LIN {X 0,Y 352.522,Z 1249.974,A -85,B 0,C 180,E1 16301.444,E2 16301.444} C_VEL
LIN {X 0,Y 352.114,Z 1252.721,A -85,B 0,C 180,E1 16297.99,E2 16297.99} C_VEL
LIN {X 0,Y 351.998,Z 1254.362,A -85,B 0,C 180,E1 16294.881,E2 16294.881} C_VEL
LIN {X 0,Y 351.964,Z 1255.218,A -85,B 0,C 180,E1 16291.783,E2 16291.783} C_VEL
LIN {X 0,Y 351.944,Z 1255.295,A -85,B 0,C 180,E1 16288.69,E2 16288.69} C_VEL
LIN {X 0,Y 351.993,Z 1254.526,A -85,B 0,C 180,E1 16285.431,E2 16285.431} C_VEL
LIN {X 0,Y 352.107,Z 1252.886,A -85,B 0,C 180,E1 16282.159,E2 16282.159} C_VEL
LIN {X 0,Y 352.483,Z 1250.205,A -85,B 0,C 180,E1 16278.706,E2 16278.706} C_VEL
LIN {X 0,Y 353.184,Z 1246.726,A -85,B 0,C 180,E1 16275.399,E2 16275.399} C_VEL
LIN {X 0,Y 354.443,Z 1242.064,A -85,B 0,C 180,E1 16271.915,E2 16271.915} C_VEL
LIN {X 0,Y 356.359,Z 1236.339,A -85,B 0,C 180,E1 16268.428,E2 16268.428} C_VEL
LIN {X 0,Y 359.376,Z 1228.818,A -85,B 0,C 180,E1 16264.623,E2 16264.623} C_VEL
LIN {X 0,Y 362.896,Z 1220.993,A -85,B 0,C 180,E1 16261.294,E2 16261.294} C_VEL
LIN {X 0,Y 363.326,Z 1218.334,A -85,B 0,C 180,E1 16260.145,E2 16260.145} C_VEL
LIN {X 0,Y 361.437,Z 1211.116,A -85,B 0,C 180,E1 16256.998,E2 16256.998} C_VEL
LIN {X 0,Y 362.2,Z 1208.382,A -85,B 0,C 180,E1 16256.041,E2 16256.041} C_VEL
LIN {X 0,Y 367.884,Z 1197.913,A -85,B 0,C 180,E1 16252.881,E2 16252.881} C_VEL
LIN {X 0,Y 374.556,Z 1185.938,A -85,B 0,C 180,E1 16249.751,E2 16249.751} C_VEL
LIN {X 0,Y 384.203,Z 1168.784,A -85,B 0,C 180,E1 16245.977,E2 16245.977} C_VEL
LIN {X 0,Y 392.178,Z 1154.367,A -85,B 0,C 180,E1 16243.302,E2 16243.302} C_VEL
LIN {X 0,Y 399.981,Z 1139.957,A -85,B 0,C 180,E1 16240.973,E2 16240.973} C_VEL
LIN {X 0,Y 408.048,Z 1124.586,A -85,B 0,C 180,E1 16238.804,E2 16238.804} C_VEL
LIN {X 0,Y 418.139,Z 1104.607,A -85,B 0,C 180,E1 16236.373,E2 16236.373} C_VEL
LIN {X 0,Y 427.575,Z 1084.304,A -85,B 0,C 180,E1 16234.304,E2 16234.304} C_VEL
LIN {X 0,Y 435.512,Z 1066.092,A -85,B 0,C 180,E1 16232.701,E2 16232.701} C_VEL
LIN {X 0,Y 442.95,Z 1047.765,A -85,B 0,C 180,E1 16231.3,E2 16231.3} C_VEL
LIN {X 0,Y 449.994,Z 1028.988,A -85,B 0,C 180,E1 16230.058,E2 16230.058} C_VEL
LIN {X 0,Y 457.896,Z 1005.714,A -85,B 0,C 180,E1 16228.73,E2 16228.73} C_VEL
LIN {X 0,Y 465.26,Z 980.582,A -85,B 0,C 180,E1 16227.557,E2 16227.557} C_VEL
LIN {X 0,Y 470.568,Z 959.738,A -85,B 0,C 180,E1 16226.745,E2 16226.745} C_VEL
LIN {X 0,Y 475.18,Z 938.773,A -85,B 0,C 180,E1 16226.067,E2 16226.067} C_VEL
LIN {X 0,Y 479.078,Z 917.527,A -85,B 0,C 180,E1 16225.5,E2 16225.5} C_VEL
LIN {X 0,Y 482.827,Z 891.865,A -85,B 0,C 180,E1 16224.963,E2 16224.963} C_VEL
LIN {X 0,Y 486.213,Z 853.496,A -85,B 0,C 180,E1 16224.337,E2 16224.337} C_VEL
LIN {X 0,Y 503.252,Z 634.163,A -85,B 0,C 180,E1 16220.941,E2 16220.941} C_VEL
LIN {X 0,Y 505.06,Z 611.125,A -85,B 0,C 180,E1 16220.573,E2 16220.573} C_VEL
LIN {X 0,Y 498.511,Z 600.707,A -85,B 0,C 180,E1 16217.962,E2 16217.962} C_VEL
LIN {X 0,Y 493.261,Z 592.705,A -85,B 0,C 180,E1 16215.52,E2 16215.52} C_VEL
LIN {X 0,Y 490.584,Z 588.712,A -85,B 0,C 180,E1 16214.097,E2 16214.097} C_VEL
LIN {X 0,Y 487.897,Z 584.679,A -85,B 0,C 180,E1 16212.487,E2 16212.487} C_VEL
LIN {X 0,Y 484.928,Z 580.257,A -85,B 0,C 180,E1 16210.398,E2 16210.398} C_VEL
LIN {X 0,Y 482.057,Z 575.835,A -85,B 0,C 180,E1 16207.808,E2 16207.808} C_VEL
LIN {X 0,Y 478.927,Z 571.053,A -85,B 0,C 180,E1 16202.872,E2 16202.872} C_VEL
LIN {X 0,Y 478.709,Z 569.893,A -85,B 0,C 180,E1 16201.676,E2 16201.676} C_VEL
LIN {X 0,Y 478.79,Z 570.06,A -85,B 0,C 180,E1 16198.325,E2 16198.325} C_VEL
LIN {X 0,Y 480.405,Z 574.169,A -85,B 0,C 180,E1 16194.506,E2 16194.506} C_VEL
LIN {X 0,Y 482.056,Z 575.82,A -85,B 0,C 180,E1 16192.611,E2 16192.611} C_VEL
LIN {X 0,Y 484.76,Z 580.113,A -85,B 0,C 180,E1 16190.142,E2 16190.142} C_VEL
LIN {X 0,Y 485.93,Z 581.746,A -85,B 0,C 180,E1 16189.268,E2 16189.268} C_VEL
LIN {X 0,Y 489.194,Z 586.617,A -85,B 0,C 180,E1 16187.127,E2 16187.127} C_VEL
LIN {X 0,Y 492.859,Z 592.145,A -85,B 0,C 180,E1 16185.099,E2 16185.099} C_VEL
LIN {X 0,Y 499.068,Z 603.052,A -85,B 0,C 180,E1 16182.149,E2 16182.149} C_VEL
LIN {X 0,Y 505.144,Z 614.212,A -85,B 0,C 180,E1 16179.695,E2 16179.695} C_VEL
LIN {X 0,Y 488.683,Z 825.696,A -85,B 0,C 180,E1 16176.415,E2 16176.415} C_VEL
LIN {X 0,Y 483.032,Z 897.393,A -85,B 0,C 180,E1 16175.281,E2 16175.281} C_VEL
LIN {X 0,Y 479.229,Z 926.302,A -85,B 0,C 180,E1 16174.732,E2 16174.732} C_VEL
LIN {X 0,Y 474.715,Z 950.697,A -85,B 0,C 180,E1 16174.14,E2 16174.14} C_VEL
LIN {X 0,Y 470.08,Z 971.607,A -85,B 0,C 180,E1 16173.509,E2 16173.509} C_VEL
LIN {X 0,Y 464.804,Z 992.221,A -85,B 0,C 180,E1 16172.758,E2 16172.758} C_VEL
LIN {X 0,Y 458.747,Z 1013.14,A -85,B 0,C 180,E1 16171.848,E2 16171.848} C_VEL
LIN {X 0,Y 450.335,Z 1038.849,A -85,B 0,C 180,E1 16170.507,E2 16170.507} C_VEL
LIN {X 0,Y 442.249,Z 1060.73,A -85,B 0,C 180,E1 16169.121,E2 16169.121} C_VEL
LIN {X 0,Y 434.787,Z 1079.328,A -85,B 0,C 180,E1 16167.755,E2 16167.755} C_VEL
LIN {X 0,Y 427.021,Z 1097.374,A -85,B 0,C 180,E1 16166.233,E2 16166.233} C_VEL
LIN {X 0,Y 418.579,Z 1115.881,A -85,B 0,C 180,E1 16164.433,E2 16164.433} C_VEL
LIN {X 0,Y 407.897,Z 1138.001,A -85,B 0,C 180,E1 16161.901,E2 16161.901} C_VEL
LIN {X 0,Y 398.718,Z 1155.96,A -85,B 0,C 180,E1 16159.457,E2 16159.457} C_VEL
LIN {X 0,Y 390.7,Z 1171.26,A -85,B 0,C 180,E1 16157.055,E2 16157.055} C_VEL
LIN {X 0,Y 382.924,Z 1185.896,A -85,B 0,C 180,E1 16154.417,E2 16154.417} C_VEL
LIN {X 0,Y 373.727,Z 1203.204,A -85,B 0,C 180,E1 16150.76,E2 16150.76} C_VEL
LIN {X 0,Y 366.731,Z 1216.395,A -85,B 0,C 180,E1 16147.452,E2 16147.452} C_VEL
LIN {X 0,Y 361.043,Z 1227.569,A -85,B 0,C 180,E1 16144.214,E2 16144.214} C_VEL
LIN {X 0,Y 356.309,Z 1237.47,A -85,B 0,C 180,E1 16140.907,E2 16140.907} C_VEL
LIN {X 0,Y 351.621,Z 1248.25,A -85,B 0,C 180,E1 16136.705,E2 16136.705} C_VEL
LIN {X 0,Y 348.103,Z 1257.41,A -85,B 0,C 180,E1 16132.288,E2 16132.288} C_VEL
LIN {X 0,Y 346.171,Z 1263.631,A -85,B 0,C 180,E1 16128.664,E2 16128.664} C_VEL
LIN {X 0,Y 344.985,Z 1268.399,A -85,B 0,C 180,E1 16125.3,E2 16125.3} C_VEL
LIN {X 0,Y 344.333,Z 1272.278,A -85,B 0,C 180,E1 16121.875,E2 16121.875} C_VEL
LIN {X 0,Y 344.037,Z 1275.131,A -85,B 0,C 180,E1 16118.531,E2 16118.531} C_VEL
LIN {X 0,Y 343.964,Z 1276.993,A -85,B 0,C 180,E1 16115.345,E2 16115.345} C_VEL
LIN {X 0,Y 343.962,Z 1278.006,A -85,B 0,C 180,E1 16112.173,E2 16112.173} C_VEL
LIN {X 0,Y 343.94,Z 1278.149,A -85,B 0,C 180,E1 16108.842,E2 16108.842} C_VEL
LIN {X 0,Y 343.96,Z 1277.351,A -85,B 0,C 180,E1 16105.506,E2 16105.506} C_VEL
LIN {X 0,Y 343.998,Z 1275.609,A -85,B 0,C 180,E1 16102.156,E2 16102.156} C_VEL
LIN {X 0,Y 344.274,Z 1272.754,A -85,B 0,C 180,E1 16098.618,E2 16098.618} C_VEL
LIN {X 0,Y 344.86,Z 1269.053,A -85,B 0,C 180,E1 16095.226,E2 16095.226} C_VEL
LIN {X 0,Y 345.976,Z 1264.369,A -85,B 0,C 180,E1 16091.822,E2 16091.822} C_VEL
LIN {X 0,Y 347.653,Z 1258.673,A -85,B 0,C 180,E1 16088.408,E2 16088.408} C_VEL
LIN {X 0,Y 350.089,Z 1251.935,A -85,B 0,C 180,E1 16085.005,E2 16085.005} C_VEL
LIN {X 0,Y 353.502,Z 1243.694,A -85,B 0,C 180,E1 16081.454,E2 16081.454} C_VEL
LIN {X 0,Y 358.794,Z 1232.318,A -85,B 0,C 180,E1 16077.284,E2 16077.284} C_VEL
LIN {X 0,Y 365.263,Z 1219.215,A -85,B 0,C 180,E1 16073.329,E2 16073.329} C_VEL
LIN {X 0,Y 371.556,Z 1207.107,A -85,B 0,C 180,E1 16070.184,E2 16070.184} C_VEL
LIN {X 0,Y 378.491,Z 1194.109,A -85,B 0,C 180,E1 16067.252,E2 16067.252} C_VEL
LIN {X 0,Y 387.733,Z 1176.97,A -85,B 0,C 180,E1 16063.924,E2 16063.924} C_VEL
LIN {X 0,Y 397.214,Z 1158.784,A -85,B 0,C 180,E1 16060.973,E2 16060.973} C_VEL
LIN {X 0,Y 405.229,Z 1143.139,A -85,B 0,C 180,E1 16058.78,E2 16058.78} C_VEL
LIN {X 0,Y 413.231,Z 1126.967,A -85,B 0,C 180,E1 16056.797,E2 16056.797} C_VEL
LIN {X 0,Y 422.005,Z 1108.433,A -85,B 0,C 180,E1 16054.822,E2 16054.822} C_VEL
LIN {X 0,Y 432.415,Z 1084.855,A -85,B 0,C 180,E1 16052.697,E2 16052.697} C_VEL
LIN {X 0,Y 440.514,Z 1064.911,A -85,B 0,C 180,E1 16051.177,E2 16051.177} C_VEL
LIN {X 0,Y 447.936,Z 1045.156,A -85,B 0,C 180,E1 16049.881,E2 16049.881} C_VEL
LIN {X 0,Y 454.93,Z 1024.851,A -85,B 0,C 180,E1 16048.74,E2 16048.74} C_VEL
LIN {X 0,Y 462.775,Z 999.429,A -85,B 0,C 180,E1 16047.541,E2 16047.541} C_VEL
LIN {X 0,Y 469.284,Z 974.478,A -85,B 0,C 180,E1 16046.594,E2 16046.594} C_VEL
LIN {X 0,Y 474.119,Z 953.034,A -85,B 0,C 180,E1 16045.932,E2 16045.932} C_VEL
LIN {X 0,Y 478.162,Z 931.716,A -85,B 0,C 180,E1 16045.396,E2 16045.396} C_VEL
LIN {X 0,Y 481.893,Z 906.777,A -85,B 0,C 180,E1 16044.891,E2 16044.891} C_VEL
LIN {X 0,Y 485.216,Z 870.124,A -85,B 0,C 180,E1 16044.283,E2 16044.283} C_VEL
LIN {X 0,Y 501.922,Z 652.969,A -85,B 0,C 180,E1 16040.912,E2 16040.912} C_VEL
LIN {X 0,Y 504.986,Z 614.146,A -85,B 0,C 180,E1 16040.304,E2 16040.304} C_VEL
LIN {X 0,Y 498.916,Z 602.978,A -85,B 0,C 180,E1 16037.856,E2 16037.856} C_VEL
LIN {X 0,Y 493.5,Z 593.583,A -85,B 0,C 180,E1 16035.332,E2 16035.332} C_VEL
LIN {X 0,Y 490.917,Z 589.346,A -85,B 0,C 180,E1 16033.967,E2 16033.967} C_VEL
LIN {X 0,Y 487.61,Z 584.438,A -85,B 0,C 180,E1 16032.013,E2 16032.013} C_VEL
LIN {X 0,Y 484.869,Z 580.341,A -85,B 0,C 180,E1 16030.095,E2 16030.095} C_VEL
LIN {X 0,Y 482.052,Z 576.133,A -85,B 0,C 180,E1 16027.629,E2 16027.629} C_VEL
LIN {X 0,Y 481.38,Z 575.198,A -85,B 0,C 180,E1 16026.919,E2 16026.919} C_VEL
LIN {X 0,Y 478.927,Z 571.706,A -85,B 0,C 180,E1 16023.231,E2 16023.231} C_VEL
LIN {X 0,Y 478.504,Z 569.885,A -85,B 0,C 180,E1 16021.557,E2 16021.557} C_VEL
LIN {X 0,Y 478.612,Z 570.097,A -85,B 0,C 180,E1 16017.485,E2 16017.485} C_VEL
LIN {X 0,Y 479.988,Z 573.755,A -85,B 0,C 180,E1 16014.261,E2 16014.261} C_VEL
LIN {X 0,Y 481.868,Z 575.726,A -85,B 0,C 180,E1 16012.068,E2 16012.068} C_VEL
LIN {X 0,Y 484.525,Z 579.925,A -85,B 0,C 180,E1 16009.657,E2 16009.657} C_VEL
LIN {X 0,Y 485.699,Z 581.553,A -85,B 0,C 180,E1 16008.782,E2 16008.782} C_VEL
LIN {X 0,Y 489.164,Z 586.725,A -85,B 0,C 180,E1 16006.525,E2 16006.525} C_VEL
LIN {X 0,Y 492.708,Z 591.978,A -85,B 0,C 180,E1 16004.583,E2 16004.583} C_VEL
LIN {X 0,Y 497.724,Z 599.573,A -85,B 0,C 180,E1 16002.22,E2 16002.22} C_VEL
LIN {X 0,Y 504.117,Z 609.822,A -85,B 0,C 180,E1 15999.629,E2 15999.629} C_VEL
LIN {X 0,Y 504.935,Z 611.35,A -85,B 0,C 180,E1 15999.316,E2 15999.316} C_VEL
LIN {X 0,Y 488.15,Z 826.267,A -85,B 0,C 180,E1 15995.989,E2 15995.989} C_VEL
LIN {X 0,Y 483.41,Z 885.211,A -85,B 0,C 180,E1 15995.055,E2 15995.055} C_VEL
LIN {X 0,Y 479.377,Z 915.107,A -85,B 0,C 180,E1 15994.461,E2 15994.461} C_VEL
LIN {X 0,Y 475.301,Z 937.602,A -85,B 0,C 180,E1 15993.871,E2 15993.871} C_VEL
LIN {X 0,Y 470.729,Z 958.575,A -85,B 0,C 180,E1 15993.198,E2 15993.198} C_VEL
LIN {X 0,Y 465.401,Z 979.63,A -85,B 0,C 180,E1 15992.385,E2 15992.385} C_VEL
LIN {X 0,Y 458.012,Z 1005.064,A -85,B 0,C 180,E1 15991.207,E2 15991.207} C_VEL
LIN {X 0,Y 450.142,Z 1028.311,A -85,B 0,C 180,E1 15989.886,E2 15989.886} C_VEL
LIN {X 0,Y 443.1,Z 1047.136,A -85,B 0,C 180,E1 15988.645,E2 15988.645} C_VEL
LIN {X 0,Y 435.599,Z 1065.66,A -85,B 0,C 180,E1 15987.234,E2 15987.234} C_VEL
LIN {X 0,Y 427.597,Z 1084.056,A -85,B 0,C 180,E1 15985.619,E2 15985.619} C_VEL
LIN {X 0,Y 417.903,Z 1104.919,A -85,B 0,C 180,E1 15983.491,E2 15983.491} C_VEL
LIN {X 0,Y 407.935,Z 1124.677,A -85,B 0,C 180,E1 15981.084,E2 15981.084} C_VEL
LIN {X 0,Y 400.126,Z 1139.578,A -85,B 0,C 180,E1 15978.983,E2 15978.983} C_VEL
LIN {X 0,Y 392.582,Z 1153.526,A -85,B 0,C 180,E1 15976.742,E2 15976.742} C_VEL
LIN {X 0,Y 384.933,Z 1167.366,A -85,B 0,C 180,E1 15974.198,E2 15974.198} C_VEL
LIN {X 0,Y 376.151,Z 1183.177,A -85,B 0,C 180,E1 15970.826,E2 15970.826} C_VEL
LIN {X 0,Y 368.306,Z 1197.109,A -85,B 0,C 180,E1 15967.247,E2 15967.247} C_VEL
LIN {X 0,Y 362.483,Z 1207.816,A -85,B 0,C 180,E1 15964.042,E2 15964.042} C_VEL
LIN {X 0,Y 357.536,Z 1217.265,A -85,B 0,C 180,E1 15960.772,E2 15960.772} C_VEL
LIN {X 0,Y 352.797,Z 1227.114,A -85,B 0,C 180,E1 15956.774,E2 15956.774} C_VEL
LIN {X 0,Y 348.985,Z 1235.881,A -85,B 0,C 180,E1 15952.39,E2 15952.39} C_VEL
LIN {X 0,Y 346.77,Z 1241.969,A -85,B 0,C 180,E1 15948.658,E2 15948.658} C_VEL
LIN {X 0,Y 345.348,Z 1246.698,A -85,B 0,C 180,E1 15945.096,E2 15945.096} C_VEL
LIN {X 0,Y 344.574,Z 1250.241,A -85,B 0,C 180,E1 15941.711,E2 15941.711} C_VEL
LIN {X 0,Y 344.136,Z 1252.986,A -85,B 0,C 180,E1 15938.177,E2 15938.177} C_VEL
LIN {X 0,Y 344.008,Z 1254.625,A -85,B 0,C 180,E1 15934.994,E2 15934.994} C_VEL
LIN {X 0,Y 343.969,Z 1255.481,A -85,B 0,C 180,E1 15931.825,E2 15931.825} C_VEL
LIN {X 0,Y 343.95,Z 1255.558,A -85,B 0,C 180,E1 15928.66,E2 15928.66} C_VEL
LIN {X 0,Y 344,Z 1254.789,A -85,B 0,C 180,E1 15925.324,E2 15925.324} C_VEL
LIN {X 0,Y 344.126,Z 1253.15,A -85,B 0,C 180,E1 15921.976,E2 15921.976} C_VEL
LIN {X 0,Y 344.532,Z 1250.471,A -85,B 0,C 180,E1 15918.441,E2 15918.441} C_VEL
LIN {X 0,Y 345.285,Z 1246.993,A -85,B 0,C 180,E1 15915.058,E2 15915.058} C_VEL
LIN {X 0,Y 346.573,Z 1242.571,A -85,B 0,C 180,E1 15911.658,E2 15911.658} C_VEL
LIN {X 0,Y 348.577,Z 1236.903,A -85,B 0,C 180,E1 15908.098,E2 15908.098} C_VEL
LIN {X 0,Y 351.424,Z 1230.118,A -85,B 0,C 180,E1 15904.549,E2 15904.549} C_VEL
LIN {X 0,Y 356.231,Z 1220.019,A -85,B 0,C 180,E1 15900.149,E2 15900.149} C_VEL
LIN {X 0,Y 361.85,Z 1209.042,A -85,B 0,C 180,E1 15896.254,E2 15896.254} C_VEL
LIN {X 0,Y 362.2,Z 1208.382,A -85,B 0,C 180,E1 15896.041,E2 15896.041} C_VEL
LIN {X 0,Y 363.073,Z 1205.259,A -85,B 0,C 180,E1 15894.93,E2 15894.93} C_VEL
LIN {X 0,Y 362.547,Z 1197.068,A -85,B 0,C 180,E1 15891.83,E2 15891.83} C_VEL
LIN {X 0,Y 363.731,Z 1194.062,A -85,B 0,C 180,E1 15890.911,E2 15890.911} C_VEL
LIN {X 0,Y 372.081,Z 1179.638,A -85,B 0,C 180,E1 15887.369,E2 15887.369} C_VEL
LIN {X 0,Y 379.545,Z 1166.783,A -85,B 0,C 180,E1 15884.653,E2 15884.653} C_VEL
LIN {X 0,Y 387.333,Z 1153.208,A -85,B 0,C 180,E1 15882.159,E2 15882.159} C_VEL
LIN {X 0,Y 395.103,Z 1139.313,A -85,B 0,C 180,E1 15879.926,E2 15879.926} C_VEL
LIN {X 0,Y 403.558,Z 1123.686,A -85,B 0,C 180,E1 15877.734,E2 15877.734} C_VEL
LIN {X 0,Y 414.629,Z 1102.104,A -85,B 0,C 180,E1 15875.158,E2 15875.158} C_VEL
LIN {X 0,Y 423.48,Z 1083.532,A -85,B 0,C 180,E1 15873.291,E2 15873.291} C_VEL
LIN {X 0,Y 431.466,Z 1065.627,A -85,B 0,C 180,E1 15871.729,E2 15871.729} C_VEL
LIN {X 0,Y 439.091,Z 1047.223,A -85,B 0,C 180,E1 15870.333,E2 15870.333} C_VEL
LIN {X 0,Y 446.971,Z 1026.569,A -85,B 0,C 180,E1 15868.987,E2 15868.987} C_VEL
LIN {X 0,Y 455.726,Z 1000.618,A -85,B 0,C 180,E1 15867.57,E2 15867.57} C_VEL
LIN {X 0,Y 461.927,Z 979.562,A -85,B 0,C 180,E1 15866.616,E2 15866.616} C_VEL
LIN {X 0,Y 467.179,Z 959.256,A -85,B 0,C 180,E1 15865.838,E2 15865.838} C_VEL
LIN {X 0,Y 471.821,Z 938.471,A -85,B 0,C 180,E1 15865.175,E2 15865.175} C_VEL
LIN {X 0,Y 475.875,Z 916.658,A -85,B 0,C 180,E1 15864.601,E2 15864.601} C_VEL
LIN {X 0,Y 479.885,Z 888.863,A -85,B 0,C 180,E1 15864.038,E2 15864.038} C_VEL
LIN {X 0,Y 483.809,Z 842.856,A -85,B 0,C 180,E1 15863.302,E2 15863.302} C_VEL
LIN {X 0,Y 501.309,Z 623.821,A -85,B 0,C 180,E1 15859.921,E2 15859.921} C_VEL
LIN {X 0,Y 501.887,Z 616.426,A -85,B 0,C 180,E1 15859.797,E2 15859.797} C_VEL
LIN {X 0,Y 495.939,Z 606.694,A -85,B 0,C 180,E1 15857.301,E2 15857.301} C_VEL
LIN {X 0,Y 490.022,Z 597.509,A -85,B 0,C 180,E1 15854.355,E2 15854.355} C_VEL
LIN {X 0,Y 486.462,Z 592.257,A -85,B 0,C 180,E1 15852.223,E2 15852.223} C_VEL
LIN {X 0,Y 483.717,Z 588.056,A -85,B 0,C 180,E1 15850.24,E2 15850.24} C_VEL
LIN {X 0,Y 480.861,Z 583.525,A -85,B 0,C 180,E1 15847.588,E2 15847.588} C_VEL
LIN {X 0,Y 477.973,Z 579.219,A -85,B 0,C 180,E1 15842.998,E2 15842.998} C_VEL
LIN {X 0,Y 477.735,Z 577.833,A -85,B 0,C 180,E1 15841.679,E2 15841.679} C_VEL
LIN {X 0,Y 477.805,Z 578.092,A -85,B 0,C 180,E1 15838.321,E2 15838.321} C_VEL
LIN {X 0,Y 479.429,Z 582.15,A -85,B 0,C 180,E1 15834.495,E2 15834.495} C_VEL
LIN {X 0,Y 480.958,Z 583.756,A -85,B 0,C 180,E1 15832.714,E2 15832.714} C_VEL
LIN {X 0,Y 483.787,Z 588.153,A -85,B 0,C 180,E1 15830.122,E2 15830.122} C_VEL
LIN {X 0,Y 487.726,Z 594.151,A -85,B 0,C 180,E1 15827.392,E2 15827.392} C_VEL
LIN {X 0,Y 491.262,Z 599.61,A -85,B 0,C 180,E1 15825.381,E2 15825.381} C_VEL
LIN {X 0,Y 497.284,Z 610.418,A -85,B 0,C 180,E1 15822.446,E2 15822.446} C_VEL
LIN {X 0,Y 501.964,Z 619.387,A -85,B 0,C 180,E1 15820.472,E2 15820.472} C_VEL
LIN {X 0,Y 484.823,Z 834.386,A -85,B 0,C 180,E1 15817.147,E2 15817.147} C_VEL
LIN {X 0,Y 479.654,Z 897.84,A -85,B 0,C 180,E1 15816.143,E2 15816.143} C_VEL
LIN {X 0,Y 475.464,Z 928.18,A -85,B 0,C 180,E1 15815.563,E2 15815.563} C_VEL
LIN {X 0,Y 471.138,Z 950.963,A -85,B 0,C 180,E1 15815.01,E2 15815.01} C_VEL
LIN {X 0,Y 466.462,Z 971.606,A -85,B 0,C 180,E1 15814.391,E2 15814.391} C_VEL
LIN {X 0,Y 460.947,Z 992.663,A -85,B 0,C 180,E1 15813.628,E2 15813.628} C_VEL
LIN {X 0,Y 453.917,Z 1016.289,A -85,B 0,C 180,E1 15812.595,E2 15812.595} C_VEL
LIN {X 0,Y 445.335,Z 1041.305,A -85,B 0,C 180,E1 15811.261,E2 15811.261} C_VEL
LIN {X 0,Y 437.699,Z 1061.412,A -85,B 0,C 180,E1 15809.98,E2 15809.98} C_VEL
LIN {X 0,Y 430.269,Z 1079.43,A -85,B 0,C 180,E1 15808.658,E2 15808.658} C_VEL
LIN {X 0,Y 422.156,Z 1097.78,A -85,B 0,C 180,E1 15807.109,E2 15807.109} C_VEL
LIN {X 0,Y 412.916,Z 1117.456,A -85,B 0,C 180,E1 15805.181,E2 15805.181} C_VEL
LIN {X 0,Y 401.692,Z 1139.783,A -85,B 0,C 180,E1 15802.572,E2 15802.572} C_VEL
LIN {X 0,Y 393.04,Z 1156.172,A -85,B 0,C 180,E1 15800.317,E2 15800.317} C_VEL
LIN {X 0,Y 384.743,Z 1171.463,A -85,B 0,C 180,E1 15797.894,E2 15797.894} C_VEL
LIN {X 0,Y 375.985,Z 1187.383,A -85,B 0,C 180,E1 15794.976,E2 15794.976} C_VEL
LIN {X 0,Y 366.62,Z 1204.223,A -85,B 0,C 180,E1 15791.307,E2 15791.307} C_VEL
LIN {X 0,Y 359.738,Z 1216.705,A -85,B 0,C 180,E1 15788.107,E2 15788.107} C_VEL
LIN {X 0,Y 354.087,Z 1227.293,A -85,B 0,C 180,E1 15784.983,E2 15784.983} C_VEL
LIN {X 0,Y 349.113,Z 1237.195,A -85,B 0,C 180,E1 15781.616,E2 15781.616} C_VEL
LIN {X 0,Y 344.038,Z 1248.264,A -85,B 0,C 180,E1 15777.209,E2 15777.209} C_VEL
LIN {X 0,Y 340.354,Z 1257.333,A -85,B 0,C 180,E1 15772.71,E2 15772.71} C_VEL
LIN {X 0,Y 338.364,Z 1263.296,A -85,B 0,C 180,E1 15769.155,E2 15769.155} C_VEL
LIN {X 0,Y 337.082,Z 1268.13,A -85,B 0,C 180,E1 15765.667,E2 15765.667} C_VEL
LIN {X 0,Y 336.377,Z 1271.981,A -85,B 0,C 180,E1 15762.191,E2 15762.191} C_VEL
LIN {X 0,Y 336.054,Z 1274.866,A -85,B 0,C 180,E1 15758.735,E2 15758.735} C_VEL
LIN {X 0,Y 335.968,Z 1276.73,A -85,B 0,C 180,E1 15755.472,E2 15755.472} C_VEL
LIN {X 0,Y 335.966,Z 1277.743,A -85,B 0,C 180,E1 15752.225,E2 15752.225} C_VEL
LIN {X 0,Y 335.946,Z 1277.886,A -85,B 0,C 180,E1 15748.814,E2 15748.814} C_VEL
LIN {X 0,Y 335.963,Z 1277.088,A -85,B 0,C 180,E1 15745.399,E2 15745.399} C_VEL
LIN {X 0,Y 336.005,Z 1275.344,A -85,B 0,C 180,E1 15741.968,E2 15741.968} C_VEL
LIN {X 0,Y 336.303,Z 1272.487,A -85,B 0,C 180,E1 15738.344,E2 15738.344} C_VEL
LIN {X 0,Y 336.935,Z 1268.783,A -85,B 0,C 180,E1 15734.871,E2 15734.871} C_VEL
LIN {X 0,Y 338.137,Z 1264.098,A -85,B 0,C 180,E1 15731.385,E2 15731.385} C_VEL
LIN {X 0,Y 339.944,Z 1258.4,A -85,B 0,C 180,E1 15727.893,E2 15727.893} C_VEL
LIN {X 0,Y 342.524,Z 1251.659,A -85,B 0,C 180,E1 15724.413,E2 15724.413} C_VEL
LIN {X 0,Y 346.138,Z 1243.417,A -85,B 0,C 180,E1 15720.789,E2 15720.789} C_VEL
LIN {X 0,Y 351.732,Z 1232.04,A -85,B 0,C 180,E1 15716.542,E2 15716.542} C_VEL
LIN {X 0,Y 358.442,Z 1219.067,A -85,B 0,C 180,E1 15712.558,E2 15712.558} C_VEL
LIN {X 0,Y 365.108,Z 1206.828,A -85,B 0,C 180,E1 15709.336,E2 15709.336} C_VEL
LIN {X 0,Y 372.332,Z 1193.83,A -85,B 0,C 180,E1 15706.37,E2 15706.37} C_VEL
LIN {X 0,Y 381.764,Z 1176.996,A -85,B 0,C 180,E1 15703.066,E2 15703.066} C_VEL
LIN {X 0,Y 391.494,Z 1158.974,A -85,B 0,C 180,E1 15700.113,E2 15700.113} C_VEL
LIN {X 0,Y 400.024,Z 1142.86,A -85,B 0,C 180,E1 15697.842,E2 15697.842} C_VEL
LIN {X 0,Y 408.279,Z 1126.689,A -85,B 0,C 180,E1 15695.858,E2 15695.858} C_VEL
LIN {X 0,Y 417.399,Z 1107.974,A -85,B 0,C 180,E1 15693.866,E2 15693.866} C_VEL
LIN {X 0,Y 428,Z 1084.579,A -85,B 0,C 180,E1 15691.765,E2 15691.765} C_VEL
LIN {X 0,Y 436.053,Z 1065.275,A -85,B 0,C 180,E1 15690.296,E2 15690.296} C_VEL
LIN {X 0,Y 443.567,Z 1045.789,A -85,B 0,C 180,E1 15689.017,E2 15689.017} C_VEL
LIN {X 0,Y 450.376,Z 1026.567,A -85,B 0,C 180,E1 15687.934,E2 15687.934} C_VEL
LIN {X 0,Y 457.059,Z 1005.7,A -85,B 0,C 180,E1 15686.927,E2 15686.927} C_VEL
LIN {X 0,Y 464.638,Z 978.662,A -85,B 0,C 180,E1 15685.853,E2 15685.853} C_VEL
LIN {X 0,Y 470.251,Z 954.609,A -85,B 0,C 180,E1 15685.098,E2 15685.098} C_VEL
LIN {X 0,Y 474.451,Z 933.191,A -85,B 0,C 180,E1 15684.557,E2 15684.557} C_VEL
LIN {X 0,Y 477.948,Z 910.895,A -85,B 0,C 180,E1 15684.1,E2 15684.1} C_VEL
LIN {X 0,Y 480.933,Z 883.238,A -85,B 0,C 180,E1 15683.619,E2 15683.619} C_VEL
LIN {X 0,Y 498.122,Z 664.777,A -85,B 0,C 180,E1 15680.235,E2 15680.235} C_VEL
LIN {X 0,Y 501.805,Z 619.102,A -85,B 0,C 180,E1 15679.519,E2 15679.519} C_VEL
LIN {X 0,Y 495.893,Z 608.046,A -85,B 0,C 180,E1 15677,E2 15677} C_VEL
LIN {X 0,Y 490.044,Z 597.708,A -85,B 0,C 180,E1 15674.052,E2 15674.052} C_VEL
LIN {X 0,Y 486.175,Z 592.008,A -85,B 0,C 180,E1 15671.748,E2 15671.748} C_VEL
LIN {X 0,Y 483.579,Z 588.063,A -85,B 0,C 180,E1 15669.882,E2 15669.882} C_VEL
LIN {X 0,Y 480.795,Z 583.696,A -85,B 0,C 180,E1 15667.348,E2 15667.348} C_VEL
LIN {X 0,Y 477.826,Z 579.278,A -85,B 0,C 180,E1 15662.879,E2 15662.879} C_VEL
LIN {X 0,Y 477.53,Z 577.825,A -85,B 0,C 180,E1 15661.56,E2 15661.56} C_VEL
LIN {X 0,Y 477.606,Z 577.985,A -85,B 0,C 180,E1 15657.6,E2 15657.6} C_VEL
LIN {X 0,Y 479.012,Z 581.749,A -85,B 0,C 180,E1 15654.25,E2 15654.25} C_VEL
LIN {X 0,Y 480.77,Z 583.665,A -85,B 0,C 180,E1 15652.17,E2 15652.17} C_VEL
LIN {X 0,Y 483.554,Z 587.969,A -85,B 0,C 180,E1 15649.636,E2 15649.636} C_VEL
LIN {X 0,Y 487.697,Z 594.269,A -85,B 0,C 180,E1 15646.785,E2 15646.785} C_VEL
LIN {X 0,Y 491.274,Z 599.696,A -85,B 0,C 180,E1 15644.778,E2 15644.778} C_VEL
LIN {X 0,Y 496.338,Z 607.575,A -85,B 0,C 180,E1 15642.351,E2 15642.351} C_VEL
LIN {X 0,Y 501.764,Z 616.409,A -85,B 0,C 180,E1 15640.099,E2 15640.099} C_VEL
LIN {X 0,Y 484.802,Z 828.429,A -85,B 0,C 180,E1 15636.824,E2 15636.824} C_VEL
LIN {X 0,Y 480.078,Z 885.602,A -85,B 0,C 180,E1 15635.92,E2 15635.92} C_VEL
LIN {X 0,Y 475.953,Z 915.514,A -85,B 0,C 180,E1 15635.328,E2 15635.328} C_VEL
LIN {X 0,Y 471.798,Z 937.985,A -85,B 0,C 180,E1 15634.743,E2 15634.743} C_VEL
LIN {X 0,Y 467.158,Z 958.849,A -85,B 0,C 180,E1 15634.078,E2 15634.078} C_VEL
LIN {X 0,Y 461.718,Z 979.903,A -85,B 0,C 180,E1 15633.272,E2 15633.272} C_VEL
LIN {X 0,Y 454.17,Z 1005.336,A -85,B 0,C 180,E1 15632.102,E2 15632.102} C_VEL
LIN {X 0,Y 446.122,Z 1028.579,A -85,B 0,C 180,E1 15630.789,E2 15630.789} C_VEL
LIN {X 0,Y 438.915,Z 1047.409,A -85,B 0,C 180,E1 15629.554,E2 15629.554} C_VEL
LIN {X 0,Y 431.298,Z 1065.784,A -85,B 0,C 180,E1 15628.158,E2 15628.158} C_VEL
LIN {X 0,Y 423.441,Z 1083.413,A -85,B 0,C 180,E1 15626.62,E2 15626.62} C_VEL
LIN {X 0,Y 413.917,Z 1103.43,A -85,B 0,C 180,E1 15624.6,E2 15624.6} C_VEL
LIN {X 0,Y 403.322,Z 1123.985,A -85,B 0,C 180,E1 15622.126,E2 15622.126} C_VEL
LIN {X 0,Y 395.163,Z 1139.089,A -85,B 0,C 180,E1 15620.006,E2 15620.006} C_VEL
LIN {X 0,Y 387.406,Z 1152.97,A -85,B 0,C 180,E1 15617.781,E2 15617.781} C_VEL
LIN {X 0,Y 379.677,Z 1166.463,A -85,B 0,C 180,E1 15615.307,E2 15615.307} C_VEL
LIN {X 0,Y 371.817,Z 1180.034,A -85,B 0,C 180,E1 15612.441,E2 15612.441} C_VEL
LIN {X 0,Y 362.484,Z 1196.053,A -85,B 0,C 180,E1 15608.427,E2 15608.427} C_VEL
LIN {X 0,Y 355.866,Z 1207.589,A -85,B 0,C 180,E1 15604.961,E2 15604.961} C_VEL
LIN {X 0,Y 350.652,Z 1217.092,A -85,B 0,C 180,E1 15601.636,E2 15601.636} C_VEL
LIN {X 0,Y 345.969,Z 1226.204,A -85,B 0,C 180,E1 15597.907,E2 15597.907} C_VEL
LIN {X 0,Y 341.508,Z 1235.859,A -85,B 0,C 180,E1 15593.09,E2 15593.09} C_VEL
LIN {X 0,Y 338.994,Z 1242.24,A -85,B 0,C 180,E1 15589.102,E2 15589.102} C_VEL
LIN {X 0,Y 337.522,Z 1246.767,A -85,B 0,C 180,E1 15585.63,E2 15585.63} C_VEL
LIN {X 0,Y 336.663,Z 1250.354,A -85,B 0,C 180,E1 15582.165,E2 15582.165} C_VEL
LIN {X 0,Y 336.182,Z 1253.142,A -85,B 0,C 180,E1 15578.544,E2 15578.544} C_VEL
LIN {X 0,Y 336.022,Z 1254.824,A -85,B 0,C 180,E1 15575.285,E2 15575.285} C_VEL
LIN {X 0,Y 335.974,Z 1255.722,A -85,B 0,C 180,E1 15572.039,E2 15572.039} C_VEL
LIN {X 0,Y 335.955,Z 1255.82,A -85,B 0,C 180,E1 15568.628,E2 15568.628} C_VEL
LIN {X 0,Y 336.005,Z 1255.117,A -85,B 0,C 180,E1 15565.384,E2 15565.384} C_VEL
LIN {X 0,Y 336.135,Z 1253.523,A -85,B 0,C 180,E1 15561.956,E2 15561.956} C_VEL
LIN {X 0,Y 336.56,Z 1250.89,A -85,B 0,C 180,E1 15558.338,E2 15558.338} C_VEL
LIN {X 0,Y 337.348,Z 1247.46,A -85,B 0,C 180,E1 15554.874,E2 15554.874} C_VEL
LIN {X 0,Y 338.789,Z 1242.847,A -85,B 0,C 180,E1 15551.227,E2 15551.227} C_VEL
LIN {X 0,Y 340.931,Z 1237.173,A -85,B 0,C 180,E1 15547.581,E2 15547.581} C_VEL
LIN {X 0,Y 343.974,Z 1230.332,A -85,B 0,C 180,E1 15543.926,E2 15543.926} C_VEL
LIN {X 0,Y 348.963,Z 1220.424,A -85,B 0,C 180,E1 15539.518,E2 15539.518} C_VEL
LIN {X 0,Y 354.946,Z 1209.314,A -85,B 0,C 180,E1 15535.506,E2 15535.506} C_VEL
LIN {X 0,Y 360.93,Z 1198.747,A -85,B 0,C 180,E1 15532.242,E2 15532.242} C_VEL
LIN {X 0,Y 363.731,Z 1194.062,A -85,B 0,C 180,E1 15530.911,E2 15530.911} C_VEL
LIN {X 0,Y 365.081,Z 1190.493,A -85,B 0,C 180,E1 15529.848,E2 15529.848} C_VEL
LIN {X 0,Y 365.794,Z 1181.177,A -85,B 0,C 180,E1 15526.857,E2 15526.857} C_VEL
LIN {X 0,Y 367.282,Z 1177.735,A -85,B 0,C 180,E1 15525.994,E2 15525.994} C_VEL
LIN {X 0,Y 375.397,Z 1164.283,A -85,B 0,C 180,E1 15523.199,E2 15523.199} C_VEL
LIN {X 0,Y 385.717,Z 1146.883,A -85,B 0,C 180,E1 15520.111,E2 15520.111} C_VEL
LIN {X 0,Y 395.945,Z 1128.663,A -85,B 0,C 180,E1 15517.422,E2 15517.422} C_VEL
LIN {X 0,Y 404.657,Z 1112.477,A -85,B 0,C 180,E1 15515.365,E2 15515.365} C_VEL
LIN {X 0,Y 413.507,Z 1095.155,A -85,B 0,C 180,E1 15513.457,E2 15513.457} C_VEL
LIN {X 0,Y 424.046,Z 1073.168,A -85,B 0,C 180,E1 15511.39,E2 15511.39} C_VEL
LIN {X 0,Y 433.716,Z 1050.703,A -85,B 0,C 180,E1 15509.635,E2 15509.635} C_VEL
LIN {X 0,Y 441.064,Z 1032.189,A -85,B 0,C 180,E1 15508.4,E2 15508.4} C_VEL
LIN {X 0,Y 447.866,Z 1013.317,A -85,B 0,C 180,E1 15507.301,E2 15507.301} C_VEL
LIN {X 0,Y 454.485,Z 993.014,A -85,B 0,C 180,E1 15506.289,E2 15506.289} C_VEL
LIN {X 0,Y 461.745,Z 967.728,A -85,B 0,C 180,E1 15505.234,E2 15505.234} C_VEL
LIN {X 0,Y 467.752,Z 942.092,A -85,B 0,C 180,E1 15504.384,E2 15504.384} C_VEL
LIN {X 0,Y 471.916,Z 920.753,A -85,B 0,C 180,E1 15503.809,E2 15503.809} C_VEL
LIN {X 0,Y 475.32,Z 899.156,A -85,B 0,C 180,E1 15503.345,E2 15503.345} C_VEL
LIN {X 0,Y 478.166,Z 874.258,A -85,B 0,C 180,E1 15502.912,E2 15502.912} C_VEL
LIN {X 0,Y 496.117,Z 654.101,A -85,B 0,C 180,E1 15499.516,E2 15499.516} C_VEL
LIN {X 0,Y 498.814,Z 621.663,A -85,B 0,C 180,E1 15499.01,E2 15499.01} C_VEL
LIN {X 0,Y 493.107,Z 612.462,A -85,B 0,C 180,E1 15496.492,E2 15496.492} C_VEL
LIN {X 0,Y 488.413,Z 604.93,A -85,B 0,C 180,E1 15494.04,E2 15494.04} C_VEL
LIN {X 0,Y 485.038,Z 599.833,A -85,B 0,C 180,E1 15491.957,E2 15491.957} C_VEL
LIN {X 0,Y 482.439,Z 595.778,A -85,B 0,C 180,E1 15490.026,E2 15490.026} C_VEL
LIN {X 0,Y 479.503,Z 591.082,A -85,B 0,C 180,E1 15487.187,E2 15487.187} C_VEL
LIN {X 0,Y 476.99,Z 587.239,A -85,B 0,C 180,E1 15483.004,E2 15483.004} C_VEL
LIN {X 0,Y 476.736,Z 585.771,A -85,B 0,C 180,E1 15481.562,E2 15481.562} C_VEL
LIN {X 0,Y 476.806,Z 585.972,A -85,B 0,C 180,E1 15478.438,E2 15478.438} C_VEL
LIN {X 0,Y 478.367,Z 590.03,A -85,B 0,C 180,E1 15474.603,E2 15474.603} C_VEL
LIN {X 0,Y 479.813,Z 591.567,A -85,B 0,C 180,E1 15472.877,E2 15472.877} C_VEL
LIN {X 0,Y 482.506,Z 595.877,A -85,B 0,C 180,E1 15470.337,E2 15470.337} C_VEL
LIN {X 0,Y 486.368,Z 601.86,A -85,B 0,C 180,E1 15467.594,E2 15467.594} C_VEL
LIN {X 0,Y 489.678,Z 607.074,A -85,B 0,C 180,E1 15465.665,E2 15465.665} C_VEL
LIN {X 0,Y 495.513,Z 617.784,A -85,B 0,C 180,E1 15462.745,E2 15462.745} C_VEL
LIN {X 0,Y 498.878,Z 624.484,A -85,B 0,C 180,E1 15461.262,E2 15461.262} C_VEL
LIN {X 0,Y 481.347,Z 839.249,A -85,B 0,C 180,E1 15457.951,E2 15457.951} C_VEL
LIN {X 0,Y 476.414,Z 897.992,A -85,B 0,C 180,E1 15457.022,E2 15457.022} C_VEL
LIN {X 0,Y 472.125,Z 928.282,A -85,B 0,C 180,E1 15456.445,E2 15456.445} C_VEL
LIN {X 0,Y 467.741,Z 950.905,A -85,B 0,C 180,E1 15455.901,E2 15455.901} C_VEL
LIN {X 0,Y 462.9,Z 971.835,A -85,B 0,C 180,E1 15455.278,E2 15455.278} C_VEL
LIN {X 0,Y 457.172,Z 993.201,A -85,B 0,C 180,E1 15454.509,E2 15454.509} C_VEL
LIN {X 0,Y 449.516,Z 1018.29,A -85,B 0,C 180,E1 15453.412,E2 15453.412} C_VEL
LIN {X 0,Y 440.758,Z 1042.855,A -85,B 0,C 180,E1 15452.087,E2 15452.087} C_VEL
LIN {X 0,Y 433.276,Z 1062.033,A -85,B 0,C 180,E1 15450.861,E2 15450.861} C_VEL
LIN {X 0,Y 425.7,Z 1079.904,A -85,B 0,C 180,E1 15449.55,E2 15449.55} C_VEL
LIN {X 0,Y 417.082,Z 1098.86,A -85,B 0,C 180,E1 15447.943,E2 15447.943} C_VEL
LIN {X 0,Y 406.438,Z 1120.814,A -85,B 0,C 180,E1 15445.758,E2 15445.758} C_VEL
LIN {X 0,Y 396.096,Z 1140.538,A -85,B 0,C 180,E1 15443.4,E2 15443.4} C_VEL
LIN {X 0,Y 387.473,Z 1156.352,A -85,B 0,C 180,E1 15441.205,E2 15441.205} C_VEL
LIN {X 0,Y 378.928,Z 1171.57,A -85,B 0,C 180,E1 15438.774,E2 15438.774} C_VEL
LIN {X 0,Y 369.297,Z 1188.479,A -85,B 0,C 180,E1 15435.633,E2 15435.633} C_VEL
LIN {X 0,Y 359.927,Z 1204.595,A -85,B 0,C 180,E1 15432.036,E2 15432.036} C_VEL
LIN {X 0,Y 352.794,Z 1217.015,A -85,B 0,C 180,E1 15428.789,E2 15428.789} C_VEL
LIN {X 0,Y 346.632,Z 1228.071,A -85,B 0,C 180,E1 15425.443,E2 15425.443} C_VEL
LIN {X 0,Y 340.565,Z 1239.758,A -85,B 0,C 180,E1 15421.31,E2 15421.31} C_VEL
LIN {X 0,Y 335.506,Z 1250.283,A -85,B 0,C 180,E1 15416.752,E2 15416.752} C_VEL
LIN {X 0,Y 332.524,Z 1257.49,A -85,B 0,C 180,E1 15413.018,E2 15413.018} C_VEL
LIN {X 0,Y 330.396,Z 1263.551,A -85,B 0,C 180,E1 15409.268,E2 15409.268} C_VEL
LIN {X 0,Y 329.044,Z 1268.439,A -85,B 0,C 180,E1 15405.572,E2 15405.572} C_VEL
LIN {X 0,Y 328.34,Z 1272.212,A -85,B 0,C 180,E1 15401.959,E2 15401.959} C_VEL
LIN {X 0,Y 328.018,Z 1275.074,A -85,B 0,C 180,E1 15398.245,E2 15398.245} C_VEL
LIN {X 0,Y 327.966,Z 1276.821,A -85,B 0,C 180,E1 15394.729,E2 15394.729} C_VEL
LIN {X 0,Y 327.952,Z 1277.622,A -85,B 0,C 180,E1 15391.231,E2 15391.231} C_VEL
LIN {X 0,Y 327.969,Z 1277.482,A -85,B 0,C 180,E1 15387.737,E2 15387.737} C_VEL
LIN {X 0,Y 327.975,Z 1276.398,A -85,B 0,C 180,E1 15384.234,E2 15384.234} C_VEL
LIN {X 0,Y 328.063,Z 1274.368,A -85,B 0,C 180,E1 15380.713,E2 15380.713} C_VEL
LIN {X 0,Y 328.532,Z 1271.057,A -85,B 0,C 180,E1 15376.814,E2 15376.814} C_VEL
LIN {X 0,Y 329.945,Z 1265.14,A -85,B 0,C 180,E1 15371.821,E2 15371.821} C_VEL
LIN {X 0,Y 332.024,Z 1258.751,A -85,B 0,C 180,E1 15367.71,E2 15367.71} C_VEL
LIN {X 0,Y 334.841,Z 1251.747,A -85,B 0,C 180,E1 15363.972,E2 15363.972} C_VEL
LIN {X 0,Y 338.417,Z 1243.971,A -85,B 0,C 180,E1 15360.445,E2 15360.445} C_VEL
LIN {X 0,Y 343.156,Z 1234.585,A -85,B 0,C 180,E1 15356.795,E2 15356.795} C_VEL
LIN {X 0,Y 350.245,Z 1221.622,A -85,B 0,C 180,E1 15352.528,E2 15352.528} C_VEL
LIN {X 0,Y 357.995,Z 1207.844,A -85,B 0,C 180,E1 15348.777,E2 15348.777} C_VEL
LIN {X 0,Y 365.426,Z 1194.977,A -85,B 0,C 180,E1 15345.767,E2 15345.767} C_VEL
LIN {X 0,Y 373.257,Z 1181.43,A -85,B 0,C 180,E1 15343.017,E2 15343.017} C_VEL
LIN {X 0,Y 383.544,Z 1163.503,A -85,B 0,C 180,E1 15339.89,E2 15339.89} C_VEL
LIN {X 0,Y 393.841,Z 1144.636,A -85,B 0,C 180,E1 15337.153,E2 15337.153} C_VEL
LIN {X 0,Y 402.571,Z 1128.097,A -85,B 0,C 180,E1 15335.091,E2 15335.091} C_VEL
LIN {X 0,Y 410.881,Z 1111.594,A -85,B 0,C 180,E1 15333.299,E2 15333.299} C_VEL
LIN {X 0,Y 419.851,Z 1092.749,A -85,B 0,C 180,E1 15331.523,E2 15331.523} C_VEL
LIN {X 0,Y 430.884,Z 1067.632,A -85,B 0,C 180,E1 15329.535,E2 15329.535} C_VEL
LIN {X 0,Y 438.959,Z 1047.328,A -85,B 0,C 180,E1 15328.191,E2 15328.191} C_VEL
LIN {X 0,Y 445.89,Z 1028.349,A -85,B 0,C 180,E1 15327.114,E2 15327.114} C_VEL
LIN {X 0,Y 452.263,Z 1009.118,A -85,B 0,C 180,E1 15326.175,E2 15326.175} C_VEL
LIN {X 0,Y 458.458,Z 988.228,A -85,B 0,C 180,E1 15325.307,E2 15325.307} C_VEL
LIN {X 0,Y 465.05,Z 962.784,A -85,B 0,C 180,E1 15324.439,E2 15324.439} C_VEL
LIN {X 0,Y 470.619,Z 935.921,A -85,B 0,C 180,E1 15323.733,E2 15323.733} C_VEL
LIN {X 0,Y 474.325,Z 913.383,A -85,B 0,C 180,E1 15323.265,E2 15323.265} C_VEL
LIN {X 0,Y 476.987,Z 890.873,A -85,B 0,C 180,E1 15322.865,E2 15322.865} C_VEL
LIN {X 0,Y 494.472,Z 675.63,A -85,B 0,C 180,E1 15319.533,E2 15319.533} C_VEL
LIN {X 0,Y 498.679,Z 624.096,A -85,B 0,C 180,E1 15318.712,E2 15318.712} C_VEL
LIN {X 0,Y 493.541,Z 614.396,A -85,B 0,C 180,E1 15316.417,E2 15316.417} C_VEL
LIN {X 0,Y 488.427,Z 605.129,A -85,B 0,C 180,E1 15313.737,E2 15313.737} C_VEL
LIN {X 0,Y 484.751,Z 599.578,A -85,B 0,C 180,E1 15311.481,E2 15311.481} C_VEL
LIN {X 0,Y 482.297,Z 595.785,A -85,B 0,C 180,E1 15309.667,E2 15309.667} C_VEL
LIN {X 0,Y 479.598,Z 591.383,A -85,B 0,C 180,E1 15307.126,E2 15307.126} C_VEL
LIN {X 0,Y 476.84,Z 587.314,A -85,B 0,C 180,E1 15302.885,E2 15302.885} C_VEL
LIN {X 0,Y 476.525,Z 585.758,A -85,B 0,C 180,E1 15301.443,E2 15301.443} C_VEL
LIN {X 0,Y 476.602,Z 585.873,A -85,B 0,C 180,E1 15297.715,E2 15297.715} C_VEL
LIN {X 0,Y 477.954,Z 589.628,A -85,B 0,C 180,E1 15294.357,E2 15294.357} C_VEL
LIN {X 0,Y 479.624,Z 591.478,A -85,B 0,C 180,E1 15292.332,E2 15292.332} C_VEL
LIN {X 0,Y 482.427,Z 595.851,A -85,B 0,C 180,E1 15289.732,E2 15289.732} C_VEL
LIN {X 0,Y 486.422,Z 602.129,A -85,B 0,C 180,E1 15286.931,E2 15286.931} C_VEL
LIN {X 0,Y 489.846,Z 607.413,A -85,B 0,C 180,E1 15284.975,E2 15284.975} C_VEL
LIN {X 0,Y 494.771,Z 615.252,A -85,B 0,C 180,E1 15282.566,E2 15282.566} C_VEL
LIN {X 0,Y 498.668,Z 621.83,A -85,B 0,C 180,E1 15280.884,E2 15280.884} C_VEL
LIN {X 0,Y 480.935,Z 838.388,A -85,B 0,C 180,E1 15277.551,E2 15277.551} C_VEL
LIN {X 0,Y 476.697,Z 887.598,A -85,B 0,C 180,E1 15276.769,E2 15276.769} C_VEL
LIN {X 0,Y 472.572,Z 916.31,A -85,B 0,C 180,E1 15276.199,E2 15276.199} C_VEL
LIN {X 0,Y 468.384,Z 938.476,A -85,B 0,C 180,E1 15275.624,E2 15275.624} C_VEL
LIN {X 0,Y 463.762,Z 958.867,A -85,B 0,C 180,E1 15274.981,E2 15274.981} C_VEL
LIN {X 0,Y 458.502,Z 978.899,A -85,B 0,C 180,E1 15274.225,E2 15274.225} C_VEL
LIN {X 0,Y 451.827,Z 1001.187,A -85,B 0,C 180,E1 15273.226,E2 15273.226} C_VEL
LIN {X 0,Y 442.89,Z 1027.066,A -85,B 0,C 180,E1 15271.819,E2 15271.819} C_VEL
LIN {X 0,Y 434.843,Z 1047.682,A -85,B 0,C 180,E1 15270.479,E2 15270.479} C_VEL
LIN {X 0,Y 427.046,Z 1066.057,A -85,B 0,C 180,E1 15269.089,E2 15269.089} C_VEL
LIN {X 0,Y 419.176,Z 1083.282,A -85,B 0,C 180,E1 15267.593,E2 15267.593} C_VEL
LIN {X 0,Y 409.981,Z 1102.106,A -85,B 0,C 180,E1 15265.71,E2 15265.71} C_VEL
LIN {X 0,Y 398.6,Z 1123.726,A -85,B 0,C 180,E1 15263.135,E2 15263.135} C_VEL
LIN {X 0,Y 389.971,Z 1139.216,A -85,B 0,C 180,E1 15260.962,E2 15260.962} C_VEL
LIN {X 0,Y 381.867,Z 1153.246,A -85,B 0,C 180,E1 15258.705,E2 15258.705} C_VEL
LIN {X 0,Y 373.555,Z 1167.265,A -85,B 0,C 180,E1 15256.111,E2 15256.111} C_VEL
LIN {X 0,Y 364.501,Z 1182.373,A -85,B 0,C 180,E1 15252.855,E2 15252.855} C_VEL
LIN {X 0,Y 355.504,Z 1197.1,A -85,B 0,C 180,E1 15249.04,E2 15249.04} C_VEL
LIN {X 0,Y 349.053,Z 1207.865,A -85,B 0,C 180,E1 15245.747,E2 15245.747} C_VEL
LIN {X 0,Y 343.595,Z 1217.367,A -85,B 0,C 180,E1 15242.364,E2 15242.364} C_VEL
LIN {X 0,Y 338.655,Z 1226.478,A -85,B 0,C 180,E1 15238.564,E2 15238.564} C_VEL
LIN {X 0,Y 333.89,Z 1236.21,A -85,B 0,C 180,E1 15233.598,E2 15233.598} C_VEL
LIN {X 0,Y 331.233,Z 1242.511,A -85,B 0,C 180,E1 15229.568,E2 15229.568} C_VEL
LIN {X 0,Y 329.637,Z 1247.121,A -85,B 0,C 180,E1 15225.937,E2 15225.937} C_VEL
LIN {X 0,Y 328.697,Z 1250.775,A -85,B 0,C 180,E1 15222.286,E2 15222.286} C_VEL
LIN {X 0,Y 328.217,Z 1253.407,A -85,B 0,C 180,E1 15218.753,E2 15218.753} C_VEL
LIN {X 0,Y 328.033,Z 1255.087,A -85,B 0,C 180,E1 15215.414,E2 15215.414} C_VEL
LIN {X 0,Y 327.979,Z 1255.984,A -85,B 0,C 180,E1 15212.088,E2 15212.088} C_VEL
LIN {X 0,Y 327.962,Z 1256.082,A -85,B 0,C 180,E1 15208.594,E2 15208.594} C_VEL
LIN {X 0,Y 328.013,Z 1255.38,A -85,B 0,C 180,E1 15205.271,E2 15205.271} C_VEL
LIN {X 0,Y 328.158,Z 1253.787,A -85,B 0,C 180,E1 15201.759,E2 15201.759} C_VEL
LIN {X 0,Y 328.616,Z 1251.156,A -85,B 0,C 180,E1 15198.052,E2 15198.052} C_VEL
LIN {X 0,Y 329.465,Z 1247.727,A -85,B 0,C 180,E1 15194.503,E2 15194.503} C_VEL
LIN {X 0,Y 331.02,Z 1243.116,A -85,B 0,C 180,E1 15190.77,E2 15190.77} C_VEL
LIN {X 0,Y 333.315,Z 1237.443,A -85,B 0,C 180,E1 15187.04,E2 15187.04} C_VEL
LIN {X 0,Y 336.507,Z 1230.661,A -85,B 0,C 180,E1 15183.334,E2 15183.334} C_VEL
LIN {X 0,Y 341.809,Z 1220.696,A -85,B 0,C 180,E1 15178.81,E2 15178.81} C_VEL
LIN {X 0,Y 348.09,Z 1209.586,A -85,B 0,C 180,E1 15174.727,E2 15174.727} C_VEL
LIN {X 0,Y 354.38,Z 1198.984,A -85,B 0,C 180,E1 15171.404,E2 15171.404} C_VEL
LIN {X 0,Y 361.204,Z 1187.727,A -85,B 0,C 180,E1 15168.359,E2 15168.359} C_VEL
LIN {X 0,Y 367.282,Z 1177.735,A -85,B 0,C 180,E1 15165.994,E2 15165.994} C_VEL
LIN {X 0,Y 369.018,Z 1173.779,A -85,B 0,C 180,E1 15164.991,E2 15164.991} C_VEL
LIN {X 0,Y 371.031,Z 1163.517,A -85,B 0,C 180,E1 15162.126,E2 15162.126} C_VEL
LIN {X 0,Y 372.818,Z 1159.718,A -85,B 0,C 180,E1 15161.331,E2 15161.331} C_VEL
LIN {X 0,Y 383.064,Z 1142.589,A -85,B 0,C 180,E1 15158.451,E2 15158.451} C_VEL
LIN {X 0,Y 391.502,Z 1128.009,A -85,B 0,C 180,E1 15156.337,E2 15156.337} C_VEL
LIN {X 0,Y 400.243,Z 1112.196,A -85,B 0,C 180,E1 15154.338,E2 15154.338} C_VEL
LIN {X 0,Y 409.343,Z 1094.819,A -85,B 0,C 180,E1 15152.435,E2 15152.435} C_VEL
LIN {X 0,Y 420.486,Z 1071.976,A -85,B 0,C 180,E1 15150.317,E2 15150.317} C_VEL
LIN {X 0,Y 429.743,Z 1050.965,A -85,B 0,C 180,E1 15148.69,E2 15148.69} C_VEL
LIN {X 0,Y 437.255,Z 1032.45,A -85,B 0,C 180,E1 15147.463,E2 15147.463} C_VEL
LIN {X 0,Y 444.208,Z 1013.576,A -85,B 0,C 180,E1 15146.372,E2 15146.372} C_VEL
LIN {X 0,Y 450.965,Z 993.272,A -85,B 0,C 180,E1 15145.369,E2 15145.369} C_VEL
LIN {X 0,Y 458.398,Z 967.864,A -85,B 0,C 180,E1 15144.319,E2 15144.319} C_VEL
LIN {X 0,Y 464.478,Z 942.42,A -85,B 0,C 180,E1 15143.483,E2 15143.483} C_VEL
LIN {X 0,Y 468.737,Z 921.002,A -85,B 0,C 180,E1 15142.912,E2 15142.912} C_VEL
LIN {X 0,Y 472.203,Z 899.402,A -85,B 0,C 180,E1 15142.452,E2 15142.452} C_VEL
LIN {X 0,Y 475.105,Z 874.498,A -85,B 0,C 180,E1 15142.023,E2 15142.023} C_VEL
LIN {X 0,Y 493.566,Z 653.554,A -85,B 0,C 180,E1 15138.627,E2 15138.627} C_VEL
LIN {X 0,Y 495.814,Z 627.096,A -85,B 0,C 180,E1 15138.215,E2 15138.215} C_VEL
LIN {X 0,Y 490.834,Z 618.895,A -85,B 0,C 180,E1 15135.902,E2 15135.902} C_VEL
LIN {X 0,Y 486.423,Z 611.788,A -85,B 0,C 180,E1 15133.492,E2 15133.492} C_VEL
LIN {X 0,Y 483.624,Z 607.408,A -85,B 0,C 180,E1 15131.69,E2 15131.69} C_VEL
LIN {X 0,Y 481.168,Z 603.499,A -85,B 0,C 180,E1 15129.811,E2 15129.811} C_VEL
LIN {X 0,Y 478.314,Z 598.881,A -85,B 0,C 180,E1 15126.964,E2 15126.964} C_VEL
LIN {X 0,Y 475.948,Z 594.978,A -85,B 0,C 180,E1 15122.77,E2 15122.77} C_VEL
LIN {X 0,Y 475.761,Z 593.711,A -85,B 0,C 180,E1 15121.566,E2 15121.566} C_VEL
LIN {X 0,Y 475.82,Z 594.002,A -85,B 0,C 180,E1 15118.435,E2 15118.435} C_VEL
LIN {X 0,Y 477.392,Z 598.011,A -85,B 0,C 180,E1 15114.592,E2 15114.592} C_VEL
LIN {X 0,Y 478.72,Z 599.497,A -85,B 0,C 180,E1 15112.982,E2 15112.982} C_VEL
LIN {X 0,Y 482.111,Z 604.953,A -85,B 0,C 180,E1 15109.846,E2 15109.846} C_VEL
LIN {X 0,Y 485.189,Z 609.874,A -85,B 0,C 180,E1 15107.684,E2 15107.684} C_VEL
LIN {X 0,Y 488.155,Z 614.641,A -85,B 0,C 180,E1 15105.922,E2 15105.922} C_VEL
LIN {X 0,Y 493.878,Z 625.371,A -85,B 0,C 180,E1 15102.989,E2 15102.989} C_VEL
LIN {X 0,Y 495.893,Z 629.517,A -85,B 0,C 180,E1 15102.063,E2 15102.063} C_VEL
LIN {X 0,Y 477.896,Z 845.006,A -85,B 0,C 180,E1 15098.752,E2 15098.752} C_VEL
LIN {X 0,Y 473.249,Z 898.536,A -85,B 0,C 180,E1 15097.906,E2 15097.906} C_VEL
LIN {X 0,Y 468.917,Z 928.291,A -85,B 0,C 180,E1 15097.341,E2 15097.341} C_VEL
LIN {X 0,Y 464.455,Z 950.865,A -85,B 0,C 180,E1 15096.804,E2 15096.804} C_VEL
LIN {X 0,Y 459.574,Z 971.578,A -85,B 0,C 180,E1 15096.195,E2 15096.195} C_VEL
LIN {X 0,Y 453.963,Z 992.145,A -85,B 0,C 180,E1 15095.466,E2 15095.466} C_VEL
LIN {X 0,Y 446.643,Z 1015.767,A -85,B 0,C 180,E1 15094.453,E2 15094.453} C_VEL
LIN {X 0,Y 437.333,Z 1041.685,A -85,B 0,C 180,E1 15093.09,E2 15093.09} C_VEL
LIN {X 0,Y 429.447,Z 1061.485,A -85,B 0,C 180,E1 15091.839,E2 15091.839} C_VEL
LIN {X 0,Y 421.569,Z 1079.636,A -85,B 0,C 180,E1 15090.519,E2 15090.519} C_VEL
LIN {X 0,Y 412.882,Z 1098.287,A -85,B 0,C 180,E1 15088.947,E2 15088.947} C_VEL
LIN {X 0,Y 402.11,Z 1119.975,A -85,B 0,C 180,E1 15086.805,E2 15086.805} C_VEL
LIN {X 0,Y 391.157,Z 1140.266,A -85,B 0,C 180,E1 15084.385,E2 15084.385} C_VEL
LIN {X 0,Y 382.112,Z 1156.348,A -85,B 0,C 180,E1 15082.146,E2 15082.146} C_VEL
LIN {X 0,Y 373.432,Z 1171.296,A -85,B 0,C 180,E1 15079.746,E2 15079.746} C_VEL
LIN {X 0,Y 363.223,Z 1188.579,A -85,B 0,C 180,E1 15076.511,E2 15076.511} C_VEL
LIN {X 0,Y 353.573,Z 1204.502,A -85,B 0,C 180,E1 15072.908,E2 15072.908} C_VEL
LIN {X 0,Y 346.246,Z 1216.739,A -85,B 0,C 180,E1 15069.665,E2 15069.665} C_VEL
LIN {X 0,Y 339.78,Z 1227.815,A -85,B 0,C 180,E1 15066.262,E2 15066.262} C_VEL
LIN {X 0,Y 333.123,Z 1240.033,A -85,B 0,C 180,E1 15061.848,E2 15061.848} C_VEL
LIN {X 0,Y 328.052,Z 1250.009,A -85,B 0,C 180,E1 15057.41,E2 15057.41} C_VEL
LIN {X 0,Y 324.777,Z 1257.473,A -85,B 0,C 180,E1 15053.443,E2 15053.443} C_VEL
LIN {X 0,Y 322.51,Z 1263.543,A -85,B 0,C 180,E1 15049.57,E2 15049.57} C_VEL
LIN {X 0,Y 321.08,Z 1268.449,A -85,B 0,C 180,E1 15045.727,E2 15045.727} C_VEL
LIN {X 0,Y 320.306,Z 1272.443,A -85,B 0,C 180,E1 15041.715,E2 15041.715} C_VEL
LIN {X 0,Y 319.999,Z 1275.701,A -85,B 0,C 180,E1 15037.007,E2 15037.007} C_VEL
LIN {X 0,Y 319.972,Z 1277.17,A -85,B 0,C 180,E1 15032.695,E2 15032.695} C_VEL
LIN {X 0,Y 319.948,Z 1277.384,A -85,B 0,C 180,E1 15028.934,E2 15028.934} C_VEL
LIN {X 0,Y 319.968,Z 1276.631,A -85,B 0,C 180,E1 15025.348,E2 15025.348} C_VEL
LIN {X 0,Y 320.018,Z 1274.932,A -85,B 0,C 180,E1 15021.745,E2 15021.745} C_VEL
LIN {X 0,Y 320.354,Z 1272.117,A -85,B 0,C 180,E1 15017.938,E2 15017.938} C_VEL
LIN {X 0,Y 321.131,Z 1268.244,A -85,B 0,C 180,E1 15014.107,E2 15014.107} C_VEL
LIN {X 0,Y 322.502,Z 1263.553,A -85,B 0,C 180,E1 15010.447,E2 15010.447} C_VEL
LIN {X 0,Y 324.773,Z 1257.457,A -85,B 0,C 180,E1 15006.558,E2 15006.558} C_VEL
LIN {X 0,Y 328.033,Z 1250.017,A -85,B 0,C 180,E1 15002.606,E2 15002.606} C_VEL
LIN {X 0,Y 333.39,Z 1239.479,A -85,B 0,C 180,E1 14997.948,E2 14997.948} C_VEL
LIN {X 0,Y 339.773,Z 1227.789,A -85,B 0,C 180,E1 14993.739,E2 14993.739} C_VEL
LIN {X 0,Y 346.209,Z 1216.752,A -85,B 0,C 180,E1 14990.35,E2 14990.35} C_VEL
LIN {X 0,Y 353.643,Z 1204.326,A -85,B 0,C 180,E1 14987.06,E2 14987.06} C_VEL
LIN {X 0,Y 363.386,Z 1188.203,A -85,B 0,C 180,E1 14983.427,E2 14983.427} C_VEL
LIN {X 0,Y 373.375,Z 1171.289,A -85,B 0,C 180,E1 14980.266,E2 14980.266} C_VEL
LIN {X 0,Y 382.205,Z 1156.068,A -85,B 0,C 180,E1 14977.824,E2 14977.824} C_VEL
LIN {X 0,Y 391.492,Z 1139.535,A -85,B 0,C 180,E1 14975.531,E2 14975.531} C_VEL
LIN {X 0,Y 402.953,Z 1118.114,A -85,B 0,C 180,E1 14973.012,E2 14973.012} C_VEL
LIN {X 0,Y 412.982,Z 1097.87,A -85,B 0,C 180,E1 14971.027,E2 14971.027} C_VEL
LIN {X 0,Y 421.487,Z 1079.576,A -85,B 0,C 180,E1 14969.487,E2 14969.487} C_VEL
LIN {X 0,Y 429.62,Z 1060.814,A -85,B 0,C 180,E1 14968.125,E2 14968.125} C_VEL
LIN {X 0,Y 437.958,Z 1039.8,A -85,B 0,C 180,E1 14966.808,E2 14966.808} C_VEL
LIN {X 0,Y 447.278,Z 1013.394,A -85,B 0,C 180,E1 14965.447,E2 14965.447} C_VEL
LIN {X 0,Y 453.874,Z 992.018,A -85,B 0,C 180,E1 14964.538,E2 14964.538} C_VEL
LIN {X 0,Y 459.485,Z 971.425,A -85,B 0,C 180,E1 14963.808,E2 14963.808} C_VEL
LIN {X 0,Y 464.442,Z 950.328,A -85,B 0,C 180,E1 14963.189,E2 14963.189} C_VEL
LIN {X 0,Y 469.069,Z 926.754,A -85,B 0,C 180,E1 14962.634,E2 14962.634} C_VEL
LIN {X 0,Y 473.262,Z 897.04,A -85,B 0,C 180,E1 14962.075,E2 14962.075} C_VEL
LIN {X 0,Y 478.981,Z 829.893,A -85,B 0,C 180,E1 14961.021,E2 14961.021} C_VEL
LIN {X 0,Y 495.746,Z 629.274,A -85,B 0,C 180,E1 14957.937,E2 14957.937} C_VEL
LIN {X 0,Y 490.575,Z 619.43,A -85,B 0,C 180,E1 14955.486,E2 14955.486} C_VEL
LIN {X 0,Y 486.824,Z 612.547,A -85,B 0,C 180,E1 14953.42,E2 14953.42} C_VEL
LIN {X 0,Y 483.422,Z 607.266,A -85,B 0,C 180,E1 14951.272,E2 14951.272} C_VEL
LIN {X 0,Y 481.171,Z 603.667,A -85,B 0,C 180,E1 14949.569,E2 14949.569} C_VEL
LIN {X 0,Y 478.455,Z 599.195,A -85,B 0,C 180,E1 14946.962,E2 14946.962} C_VEL
LIN {X 0,Y 475.82,Z 595.194,A -85,B 0,C 180,E1 14942.77,E2 14942.77} C_VEL
LIN {X 0,Y 475.523,Z 593.69,A -85,B 0,C 180,E1 14941.325,E2 14941.325} C_VEL
LIN {X 0,Y 475.613,Z 593.931,A -85,B 0,C 180,E1 14937.711,E2 14937.711} C_VEL
LIN {X 0,Y 477.143,Z 597.839,A -85,B 0,C 180,E1 14934.106,E2 14934.106} C_VEL
LIN {X 0,Y 478.53,Z 599.41,A -85,B 0,C 180,E1 14932.436,E2 14932.436} C_VEL
LIN {X 0,Y 481.881,Z 604.773,A -85,B 0,C 180,E1 14929.358,E2 14929.358} C_VEL
LIN {X 0,Y 485.152,Z 609.984,A -85,B 0,C 180,E1 14927.078,E2 14927.078} C_VEL
LIN {X 0,Y 488.53,Z 615.296,A -85,B 0,C 180,E1 14925.116,E2 14925.116} C_VEL
LIN {X 0,Y 493.953,Z 624.138,A -85,B 0,C 180,E1 14922.445,E2 14922.445} C_VEL
LIN {X 0,Y 495.659,Z 627.269,A -85,B 0,C 180,E1 14921.679,E2 14921.679} C_VEL
LIN {X 0,Y 477.556,Z 843.322,A -85,B 0,C 180,E1 14918.366,E2 14918.366} C_VEL
LIN {X 0,Y 473.447,Z 889.357,A -85,B 0,C 180,E1 14917.635,E2 14917.635} C_VEL
LIN {X 0,Y 469.301,Z 917.106,A -85,B 0,C 180,E1 14917.082,E2 14917.082} C_VEL
LIN {X 0,Y 465.082,Z 938.967,A -85,B 0,C 180,E1 14916.519,E2 14916.519} C_VEL
LIN {X 0,Y 460.384,Z 959.281,A -85,B 0,C 180,E1 14915.883,E2 14915.883} C_VEL
LIN {X 0,Y 455.054,Z 979.172,A -85,B 0,C 180,E1 14915.139,E2 14915.139} C_VEL
LIN {X 0,Y 448.244,Z 1001.46,A -85,B 0,C 180,E1 14914.148,E2 14914.148} C_VEL
LIN {X 0,Y 439.21,Z 1027.088,A -85,B 0,C 180,E1 14912.768,E2 14912.768} C_VEL
LIN {X 0,Y 430.89,Z 1047.954,A -85,B 0,C 180,E1 14911.421,E2 14911.421} C_VEL
LIN {X 0,Y 422.911,Z 1066.33,A -85,B 0,C 180,E1 14910.038,E2 14910.038} C_VEL
LIN {X 0,Y 414.841,Z 1083.556,A -85,B 0,C 180,E1 14908.549,E2 14908.549} C_VEL
LIN {X 0,Y 405.071,Z 1103.039,A -85,B 0,C 180,E1 14906.601,E2 14906.601} C_VEL
LIN {X 0,Y 393.541,Z 1124.272,A -85,B 0,C 180,E1 14904.061,E2 14904.061} C_VEL
LIN {X 0,Y 384.8,Z 1139.491,A -85,B 0,C 180,E1 14901.922,E2 14901.922} C_VEL
LIN {X 0,Y 376.077,Z 1154.108,A -85,B 0,C 180,E1 14899.554,E2 14899.554} C_VEL
LIN {X 0,Y 367.441,Z 1168.177,A -85,B 0,C 180,E1 14896.919,E2 14896.919} C_VEL
LIN {X 0,Y 357.607,Z 1184.004,A -85,B 0,C 180,E1 14893.445,E2 14893.445} C_VEL
LIN {X 0,Y 348.703,Z 1197.937,A -85,B 0,C 180,E1 14889.738,E2 14889.738} C_VEL
LIN {X 0,Y 342.002,Z 1208.644,A -85,B 0,C 180,E1 14886.394,E2 14886.394} C_VEL
LIN {X 0,Y 336.326,Z 1218.089,A -85,B 0,C 180,E1 14882.949,E2 14882.949} C_VEL
LIN {X 0,Y 330.558,Z 1228.329,A -85,B 0,C 180,E1 14878.539,E2 14878.539} C_VEL
LIN {X 0,Y 326.077,Z 1236.991,A -85,B 0,C 180,E1 14873.866,E2 14873.866} C_VEL
LIN {X 0,Y 323.459,Z 1242.868,A -85,B 0,C 180,E1 14869.992,E2 14869.992} C_VEL
LIN {X 0,Y 321.738,Z 1247.543,A -85,B 0,C 180,E1 14866.197,E2 14866.197} C_VEL
LIN {X 0,Y 320.768,Z 1251.042,A -85,B 0,C 180,E1 14862.594,E2 14862.594} C_VEL
LIN {X 0,Y 320.249,Z 1253.672,A -85,B 0,C 180,E1 14858.972,E2 14858.972} C_VEL
LIN {X 0,Y 320.044,Z 1255.351,A -85,B 0,C 180,E1 14855.549,E2 14855.549} C_VEL
LIN {X 0,Y 319.983,Z 1256.247,A -85,B 0,C 180,E1 14852.141,E2 14852.141} C_VEL
LIN {X 0,Y 319.958,Z 1256.367,A -85,B 0,C 180,E1 14848.738,E2 14848.738} C_VEL
LIN {X 0,Y 320.02,Z 1255.643,A -85,B 0,C 180,E1 14845.153,E2 14845.153} C_VEL
LIN {X 0,Y 320.184,Z 1254.052,A -85,B 0,C 180,E1 14841.552,E2 14841.552} C_VEL
LIN {X 0,Y 320.68,Z 1251.422,A -85,B 0,C 180,E1 14837.751,E2 14837.751} C_VEL
LIN {X 0,Y 321.598,Z 1247.995,A -85,B 0,C 180,E1 14834.114,E2 14834.114} C_VEL
LIN {X 0,Y 323.267,Z 1243.385,A -85,B 0,C 180,E1 14830.29,E2 14830.29} C_VEL
LIN {X 0,Y 325.731,Z 1237.713,A -85,B 0,C 180,E1 14826.473,E2 14826.473} C_VEL
LIN {X 0,Y 329.11,Z 1230.932,A -85,B 0,C 180,E1 14822.685,E2 14822.685} C_VEL
LIN {X 0,Y 334.713,Z 1220.968,A -85,B 0,C 180,E1 14818.072,E2 14818.072} C_VEL
LIN {X 0,Y 341.298,Z 1209.859,A -85,B 0,C 180,E1 14813.917,E2 14813.917} C_VEL
LIN {X 0,Y 347.871,Z 1199.291,A -85,B 0,C 180,E1 14810.556,E2 14810.556} C_VEL
LIN {X 0,Y 355.016,Z 1187.998,A -85,B 0,C 180,E1 14807.465,E2 14807.465} C_VEL
LIN {X 0,Y 364.374,Z 1173.302,A -85,B 0,C 180,E1 14804.024,E2 14804.024} C_VEL
LIN {X 0,Y 372.818,Z 1159.718,A -85,B 0,C 180,E1 14801.331,E2 14801.331} C_VEL
LIN {X 0,Y 374.859,Z 1155.258,A -85,B 0,C 180,E1 14800.412,E2 14800.412} C_VEL
LIN {X 0,Y 377.569,Z 1144.541,A -85,B 0,C 180,E1 14797.853,E2 14797.853} C_VEL
LIN {X 0,Y 379.831,Z 1139.752,A -85,B 0,C 180,E1 14796.987,E2 14796.987} C_VEL
LIN {X 0,Y 391.145,Z 1120.656,A -85,B 0,C 180,E1 14794.335,E2 14794.335} C_VEL
LIN {X 0,Y 402.48,Z 1099.867,A -85,B 0,C 180,E1 14791.949,E2 14791.949} C_VEL
LIN {X 0,Y 411.464,Z 1082.344,A -85,B 0,C 180,E1 14790.237,E2 14790.237} C_VEL
LIN {X 0,Y 419.797,Z 1064.916,A -85,B 0,C 180,E1 14788.76,E2 14788.76} C_VEL
LIN {X 0,Y 428.223,Z 1045.814,A -85,B 0,C 180,E1 14787.353,E2 14787.353} C_VEL
LIN {X 0,Y 438.526,Z 1019.822,A -85,B 0,C 180,E1 14785.75,E2 14785.75} C_VEL
LIN {X 0,Y 446.128,Z 997.939,A -85,B 0,C 180,E1 14784.638,E2 14784.638} C_VEL
LIN {X 0,Y 452.344,Z 977.776,A -85,B 0,C 180,E1 14783.769,E2 14783.769} C_VEL
LIN {X 0,Y 457.797,Z 957.587,A -85,B 0,C 180,E1 14783.033,E2 14783.033} C_VEL
LIN {X 0,Y 463.118,Z 934.499,A -85,B 0,C 180,E1 14782.336,E2 14782.336} C_VEL
LIN {X 0,Y 468.342,Z 905.573,A -85,B 0,C 180,E1 14781.662,E2 14781.662} C_VEL
LIN {X 0,Y 471.37,Z 882.301,A -85,B 0,C 180,E1 14781.246,E2 14781.246} C_VEL
LIN {X 0,Y 489.205,Z 675.035,A -85,B 0,C 180,E1 14778.063,E2 14778.063} C_VEL
LIN {X 0,Y 492.932,Z 632.472,A -85,B 0,C 180,E1 14777.416,E2 14777.416} C_VEL
LIN {X 0,Y 487.231,Z 623.05,A -85,B 0,C 180,E1 14774.56,E2 14774.56} C_VEL
LIN {X 0,Y 482.993,Z 616.008,A -85,B 0,C 180,E1 14771.948,E2 14771.948} C_VEL
LIN {X 0,Y 479.904,Z 611.218,A -85,B 0,C 180,E1 14769.595,E2 14769.595} C_VEL
LIN {X 0,Y 477.236,Z 606.765,A -85,B 0,C 180,E1 14766.859,E2 14766.859} C_VEL
LIN {X 0,Y 474.938,Z 602.857,A -85,B 0,C 180,E1 14762.655,E2 14762.655} C_VEL
LIN {X 0,Y 474.764,Z 601.649,A -85,B 0,C 180,E1 14761.448,E2 14761.448} C_VEL
LIN {X 0,Y 474.823,Z 601.881,A -85,B 0,C 180,E1 14758.552,E2 14758.552} C_VEL
LIN {X 0,Y 476.332,Z 605.891,A -85,B 0,C 180,E1 14754.7,E2 14754.7} C_VEL
LIN {X 0,Y 477.629,Z 607.425,A -85,B 0,C 180,E1 14753.086,E2 14753.086} C_VEL
LIN {X 0,Y 480.897,Z 612.779,A -85,B 0,C 180,E1 14750.002,E2 14750.002} C_VEL
LIN {X 0,Y 483.835,Z 617.572,A -85,B 0,C 180,E1 14747.892,E2 14747.892} C_VEL
LIN {X 0,Y 486.593,Z 622.105,A -85,B 0,C 180,E1 14746.21,E2 14746.21} C_VEL
LIN {X 0,Y 492.191,Z 632.848,A -85,B 0,C 180,E1 14743.264,E2 14743.264} C_VEL
LIN {X 0,Y 492.988,Z 634.757,A -85,B 0,C 180,E1 14742.871,E2 14742.871} C_VEL
LIN {X 0,Y 474.559,Z 850.507,A -85,B 0,C 180,E1 14739.568,E2 14739.568} C_VEL
LIN {X 0,Y 470.155,Z 899.5,A -85,B 0,C 180,E1 14738.796,E2 14738.796} C_VEL
LIN {X 0,Y 465.8,Z 928.431,A -85,B 0,C 180,E1 14738.246,E2 14738.246} C_VEL
LIN {X 0,Y 461.295,Z 950.787,A -85,B 0,C 180,E1 14737.722,E2 14737.722} C_VEL
LIN {X 0,Y 456.367,Z 971.321,A -85,B 0,C 180,E1 14737.124,E2 14737.124} C_VEL
LIN {X 0,Y 450.651,Z 991.886,A -85,B 0,C 180,E1 14736.405,E2 14736.405} C_VEL
LIN {X 0,Y 443.188,Z 1015.506,A -85,B 0,C 180,E1 14735.405,E2 14735.405} C_VEL
LIN {X 0,Y 433.685,Z 1041.421,A -85,B 0,C 180,E1 14734.056,E2 14734.056} C_VEL
LIN {X 0,Y 425.532,Z 1061.434,A -85,B 0,C 180,E1 14732.802,E2 14732.802} C_VEL
LIN {X 0,Y 417.222,Z 1080.111,A -85,B 0,C 180,E1 14731.449,E2 14731.449} C_VEL
LIN {X 0,Y 407.861,Z 1099.672,A -85,B 0,C 180,E1 14729.795,E2 14729.795} C_VEL
LIN {X 0,Y 395.415,Z 1123.642,A -85,B 0,C 180,E1 14727.365,E2 14727.365} C_VEL
LIN {X 0,Y 385.528,Z 1141.412,A -85,B 0,C 180,E1 14725.209,E2 14725.209} C_VEL
LIN {X 0,Y 376.482,Z 1156.983,A -85,B 0,C 180,E1 14723.018,E2 14723.018} C_VEL
LIN {X 0,Y 366.658,Z 1173.337,A -85,B 0,C 180,E1 14720.347,E2 14720.347} C_VEL
LIN {X 0,Y 355.367,Z 1191.567,A -85,B 0,C 180,E1 14716.788,E2 14716.788} C_VEL
LIN {X 0,Y 346.719,Z 1205.338,A -85,B 0,C 180,E1 14713.577,E2 14713.577} C_VEL
LIN {X 0,Y 339.415,Z 1217.048,A -85,B 0,C 180,E1 14710.406,E2 14710.406} C_VEL
LIN {X 0,Y 332.403,Z 1228.573,A -85,B 0,C 180,E1 14706.777,E2 14706.777} C_VEL
LIN {X 0,Y 324.834,Z 1241.744,A -85,B 0,C 180,E1 14701.768,E2 14701.768} C_VEL
LIN {X 0,Y 320.268,Z 1250.462,A -85,B 0,C 180,E1 14697.73,E2 14697.73} C_VEL
LIN {X 0,Y 316.993,Z 1257.571,A -85,B 0,C 180,E1 14693.82,E2 14693.82} C_VEL
LIN {X 0,Y 314.546,Z 1263.798,A -85,B 0,C 180,E1 14689.699,E2 14689.699} C_VEL
LIN {X 0,Y 312.89,Z 1269.464,A -85,B 0,C 180,E1 14685.009,E2 14685.009} C_VEL
LIN {X 0,Y 312.142,Z 1273.476,A -85,B 0,C 180,E1 14680.342,E2 14680.342} C_VEL
LIN {X 0,Y 311.991,Z 1275.796,A -85,B 0,C 180,E1 14676.264,E2 14676.264} C_VEL
LIN {X 0,Y 311.976,Z 1276.932,A -85,B 0,C 180,E1 14672.58,E2 14672.58} C_VEL
LIN {X 0,Y 311.953,Z 1277.121,A -85,B 0,C 180,E1 14668.906,E2 14668.906} C_VEL
LIN {X 0,Y 311.971,Z 1276.368,A -85,B 0,C 180,E1 14665.229,E2 14665.229} C_VEL
LIN {X 0,Y 312.035,Z 1274.667,A -85,B 0,C 180,E1 14661.533,E2 14661.533} C_VEL
LIN {X 0,Y 312.397,Z 1271.85,A -85,B 0,C 180,E1 14657.626,E2 14657.626} C_VEL
LIN {X 0,Y 313.251,Z 1267.974,A -85,B 0,C 180,E1 14653.696,E2 14653.696} C_VEL
LIN {X 0,Y 314.72,Z 1263.281,A -85,B 0,C 180,E1 14649.943,E2 14649.943} C_VEL
LIN {X 0,Y 317.113,Z 1257.266,A -85,B 0,C 180,E1 14646.01,E2 14646.01} C_VEL
LIN {X 0,Y 320.62,Z 1249.741,A -85,B 0,C 180,E1 14641.918,E2 14641.918} C_VEL
LIN {X 0,Y 326.282,Z 1239.201,A -85,B 0,C 180,E1 14637.164,E2 14637.164} C_VEL
LIN {X 0,Y 332.995,Z 1227.533,A -85,B 0,C 180,E1 14632.888,E2 14632.888} C_VEL
LIN {X 0,Y 339.735,Z 1216.473,A -85,B 0,C 180,E1 14629.439,E2 14629.439} C_VEL
LIN {X 0,Y 347.489,Z 1204.046,A -85,B 0,C 180,E1 14626.108,E2 14626.108} C_VEL
LIN {X 0,Y 357.634,Z 1187.924,A -85,B 0,C 180,E1 14622.444,E2 14622.444} C_VEL
LIN {X 0,Y 367.992,Z 1171.011,A -85,B 0,C 180,E1 14619.266,E2 14619.266} C_VEL
LIN {X 0,Y 377.14,Z 1155.754,A -85,B 0,C 180,E1 14616.812,E2 14616.812} C_VEL
LIN {X 0,Y 386.572,Z 1139.457,A -85,B 0,C 180,E1 14614.548,E2 14614.548} C_VEL
LIN {X 0,Y 398.165,Z 1118.452,A -85,B 0,C 180,E1 14612.072,E2 14612.072} C_VEL
LIN {X 0,Y 408.77,Z 1097.593,A -85,B 0,C 180,E1 14610.031,E2 14610.031} C_VEL
LIN {X 0,Y 417.479,Z 1079.3,A -85,B 0,C 180,E1 14608.499,E2 14608.499} C_VEL
LIN {X 0,Y 425.799,Z 1060.539,A -85,B 0,C 180,E1 14607.148,E2 14607.148} C_VEL
LIN {X 0,Y 434.323,Z 1039.525,A -85,B 0,C 180,E1 14605.843,E2 14605.843} C_VEL
LIN {X 0,Y 443.915,Z 1012.871,A -85,B 0,C 180,E1 14604.485,E2 14604.485} C_VEL
LIN {X 0,Y 450.77,Z 991.034,A -85,B 0,C 180,E1 14603.571,E2 14603.571} C_VEL
LIN {X 0,Y 456.47,Z 970.408,A -85,B 0,C 180,E1 14602.855,E2 14602.855} C_VEL
LIN {X 0,Y 461.581,Z 948.888,A -85,B 0,C 180,E1 14602.236,E2 14602.236} C_VEL
LIN {X 0,Y 466.879,Z 921.858,A -85,B 0,C 180,E1 14601.623,E2 14601.623} C_VEL
LIN {X 0,Y 470.489,Z 894.856,A -85,B 0,C 180,E1 14601.134,E2 14601.134} C_VEL
LIN {X 0,Y 482.617,Z 752.931,A -85,B 0,C 180,E1 14598.94,E2 14598.94} C_VEL
LIN {X 0,Y 492.803,Z 634.369,A -85,B 0,C 180,E1 14597.11,E2 14597.11} C_VEL
LIN {X 0,Y 488.043,Z 625.155,A -85,B 0,C 180,E1 14594.717,E2 14594.717} C_VEL
LIN {X 0,Y 485.138,Z 619.823,A -85,B 0,C 180,E1 14593.043,E2 14593.043} C_VEL
LIN {X 0,Y 482.017,Z 614.833,A -85,B 0,C 180,E1 14591.002,E2 14591.002} C_VEL
LIN {X 0,Y 479.899,Z 611.387,A -85,B 0,C 180,E1 14589.353,E2 14589.353} C_VEL
LIN {X 0,Y 477.05,Z 606.73,A -85,B 0,C 180,E1 14586.499,E2 14586.499} C_VEL
LIN {X 0,Y 474.802,Z 603.074,A -85,B 0,C 180,E1 14582.655,E2 14582.655} C_VEL
LIN {X 0,Y 474.548,Z 601.63,A -85,B 0,C 180,E1 14581.328,E2 14581.328} C_VEL
LIN {X 0,Y 474.611,Z 601.817,A -85,B 0,C 180,E1 14577.827,E2 14577.827} C_VEL
LIN {X 0,Y 476.168,Z 605.825,A -85,B 0,C 180,E1 14574.094,E2 14574.094} C_VEL
LIN {X 0,Y 477.439,Z 607.339,A -85,B 0,C 180,E1 14572.539,E2 14572.539} C_VEL
LIN {X 0,Y 480.596,Z 612.464,A -85,B 0,C 180,E1 14569.572,E2 14569.572} C_VEL
LIN {X 0,Y 483.795,Z 617.683,A -85,B 0,C 180,E1 14567.284,E2 14567.284} C_VEL
LIN {X 0,Y 487.324,Z 623.339,A -85,B 0,C 180,E1 14565.2,E2 14565.2} C_VEL
LIN {X 0,Y 492.77,Z 632.399,A -85,B 0,C 180,E1 14562.49,E2 14562.49} C_VEL
LIN {X 0,Y 474.458,Z 846.069,A -85,B 0,C 180,E1 14559.227,E2 14559.227} C_VEL
LIN {X 0,Y 470.337,Z 890.817,A -85,B 0,C 180,E1 14558.517,E2 14558.517} C_VEL
LIN {X 0,Y 466.12,Z 918.032,A -85,B 0,C 180,E1 14557.974,E2 14557.974} C_VEL
LIN {X 0,Y 461.847,Z 939.673,A -85,B 0,C 180,E1 14557.42,E2 14557.42} C_VEL
LIN {X 0,Y 456.922,Z 960.48,A -85,B 0,C 180,E1 14556.771,E2 14556.771} C_VEL
LIN {X 0,Y 450.991,Z 981.999,A -85,B 0,C 180,E1 14555.964,E2 14555.964} C_VEL
LIN {X 0,Y 442.241,Z 1009.146,A -85,B 0,C 180,E1 14554.719,E2 14554.719} C_VEL
LIN {X 0,Y 434.395,Z 1030.29,A -85,B 0,C 180,E1 14553.539,E2 14553.539} C_VEL
LIN {X 0,Y 426.709,Z 1049.031,A -85,B 0,C 180,E1 14552.324,E2 14552.324} C_VEL
LIN {X 0,Y 418.558,Z 1067.33,A -85,B 0,C 180,E1 14550.947,E2 14550.947} C_VEL
LIN {X 0,Y 409.976,Z 1085.151,A -85,B 0,C 180,E1 14549.403,E2 14549.403} C_VEL
LIN {X 0,Y 398.573,Z 1107.111,A -85,B 0,C 180,E1 14547.166,E2 14547.166} C_VEL
LIN {X 0,Y 388.028,Z 1125.776,A -85,B 0,C 180,E1 14544.883,E2 14544.883} C_VEL
LIN {X 0,Y 379.189,Z 1140.679,A -85,B 0,C 180,E1 14542.767,E2 14542.767} C_VEL
LIN {X 0,Y 370.327,Z 1155.043,A -85,B 0,C 180,E1 14540.416,E2 14540.416} C_VEL
LIN {X 0,Y 360.633,Z 1170.321,A -85,B 0,C 180,E1 14537.505,E2 14537.505} C_VEL
LIN {X 0,Y 349.664,Z 1187.098,A -85,B 0,C 180,E1 14533.658,E2 14533.658} C_VEL
LIN {X 0,Y 341.582,Z 1199.335,A -85,B 0,C 180,E1 14530.297,E2 14530.297} C_VEL
LIN {X 0,Y 334.999,Z 1209.423,A -85,B 0,C 180,E1 14527.067,E2 14527.067} C_VEL
LIN {X 0,Y 328.822,Z 1219.259,A -85,B 0,C 180,E1 14523.382,E2 14523.382} C_VEL
LIN {X 0,Y 322.234,Z 1230.364,A -85,B 0,C 180,E1 14518.332,E2 14518.332} C_VEL
LIN {X 0,Y 318.23,Z 1237.851,A -85,B 0,C 180,E1 14514.098,E2 14514.098} C_VEL
LIN {X 0,Y 315.566,Z 1243.544,A -85,B 0,C 180,E1 14510.194,E2 14510.194} C_VEL
LIN {X 0,Y 313.843,Z 1247.972,A -85,B 0,C 180,E1 14506.463,E2 14506.463} C_VEL
LIN {X 0,Y 312.805,Z 1251.463,A -85,B 0,C 180,E1 14502.733,E2 14502.733} C_VEL
LIN {X 0,Y 312.262,Z 1254.046,A -85,B 0,C 180,E1 14499.018,E2 14499.018} C_VEL
LIN {X 0,Y 312.048,Z 1255.68,A -85,B 0,C 180,E1 14495.508,E2 14495.508} C_VEL
LIN {X 0,Y 311.988,Z 1256.531,A -85,B 0,C 180,E1 14492.012,E2 14492.012} C_VEL
LIN {X 0,Y 311.972,Z 1256.607,A -85,B 0,C 180,E1 14488.522,E2 14488.522} C_VEL
LIN {X 0,Y 312.027,Z 1255.906,A -85,B 0,C 180,E1 14485.028,E2 14485.028} C_VEL
LIN {X 0,Y 312.212,Z 1254.316,A -85,B 0,C 180,E1 14481.335,E2 14481.335} C_VEL
LIN {X 0,Y 312.75,Z 1251.688,A -85,B 0,C 180,E1 14477.436,E2 14477.436} C_VEL
LIN {X 0,Y 313.747,Z 1248.262,A -85,B 0,C 180,E1 14473.705,E2 14473.705} C_VEL
LIN {X 0,Y 315.534,Z 1243.654,A -85,B 0,C 180,E1 14469.786,E2 14469.786} C_VEL
LIN {X 0,Y 318.177,Z 1237.983,A -85,B 0,C 180,E1 14465.88,E2 14465.88} C_VEL
LIN {X 0,Y 321.96,Z 1230.86,A -85,B 0,C 180,E1 14461.825,E2 14461.825} C_VEL
LIN {X 0,Y 328.288,Z 1220.197,A -85,B 0,C 180,E1 14456.887,E2 14456.887} C_VEL
LIN {X 0,Y 334.897,Z 1209.628,A -85,B 0,C 180,E1 14452.9,E2 14452.9} C_VEL
LIN {X 0,Y 341.842,Z 1199.002,A -85,B 0,C 180,E1 14449.5,E2 14449.5} C_VEL
LIN {X 0,Y 349.766,Z 1187.024,A -85,B 0,C 180,E1 14446.219,E2 14446.219} C_VEL
LIN {X 0,Y 360.981,Z 1169.867,A -85,B 0,C 180,E1 14442.298,E2 14442.298} C_VEL
LIN {X 0,Y 369.942,Z 1155.789,A -85,B 0,C 180,E1 14439.612,E2 14439.612} C_VEL
LIN {X 0,Y 379.213,Z 1140.773,A -85,B 0,C 180,E1 14437.144,E2 14437.144} C_VEL
LIN {X 0,Y 379.831,Z 1139.752,A -85,B 0,C 180,E1 14436.987,E2 14436.987} C_VEL
LIN {X 0,Y 382.165,Z 1134.999,A -85,B 0,C 180,E1 14436.136,E2 14436.136} C_VEL
LIN {X 0,Y 386.004,Z 1122.568,A -85,B 0,C 180,E1 14433.627,E2 14433.627} C_VEL
LIN {X 0,Y 388.156,Z 1118.069,A -85,B 0,C 180,E1 14432.977,E2 14432.977} C_VEL
LIN {X 0,Y 398.496,Z 1099.561,A -85,B 0,C 180,E1 14430.885,E2 14430.885} C_VEL
LIN {X 0,Y 407.729,Z 1081.948,A -85,B 0,C 180,E1 14429.18,E2 14429.18} C_VEL
LIN {X 0,Y 416.601,Z 1063.768,A -85,B 0,C 180,E1 14427.662,E2 14427.662} C_VEL
LIN {X 0,Y 426.801,Z 1041.005,A -85,B 0,C 180,E1 14426.039,E2 14426.039} C_VEL
LIN {X 0,Y 435.999,Z 1017.517,A -85,B 0,C 180,E1 14424.651,E2 14424.651} C_VEL
LIN {X 0,Y 443.164,Z 997.157,A -85,B 0,C 180,E1 14423.639,E2 14423.639} C_VEL
LIN {X 0,Y 449.4,Z 977.208,A -85,B 0,C 180,E1 14422.796,E2 14422.796} C_VEL
LIN {X 0,Y 455.226,Z 955.855,A -85,B 0,C 180,E1 14422.035,E2 14422.035} C_VEL
LIN {X 0,Y 461.43,Z 928.569,A -85,B 0,C 180,E1 14421.251,E2 14421.251} C_VEL
LIN {X 0,Y 465.768,Z 903.617,A -85,B 0,C 180,E1 14420.703,E2 14420.703} C_VEL
LIN {X 0,Y 468.661,Z 881.28,A -85,B 0,C 180,E1 14420.312,E2 14420.312} C_VEL
LIN {X 0,Y 487.417,Z 668.143,A -85,B 0,C 180,E1 14417.059,E2 14417.059} C_VEL
LIN {X 0,Y 490.097,Z 638.035,A -85,B 0,C 180,E1 14416.596,E2 14416.596} C_VEL
LIN {X 0,Y 485.218,Z 629.745,A -85,B 0,C 180,E1 14414.013,E2 14414.013} C_VEL
LIN {X 0,Y 481.156,Z 623.023,A -85,B 0,C 180,E1 14411.386,E2 14411.386} C_VEL
LIN {X 0,Y 478.787,Z 619.103,A -85,B 0,C 180,E1 14409.496,E2 14409.496} C_VEL
LIN {X 0,Y 476.058,Z 614.56,A -85,B 0,C 180,E1 14406.634,E2 14406.634} C_VEL
LIN {X 0,Y 473.907,Z 610.595,A -85,B 0,C 180,E1 14402.419,E2 14402.419} C_VEL
LIN {X 0,Y 473.769,Z 609.587,A -85,B 0,C 180,E1 14401.33,E2 14401.33} C_VEL
LIN {X 0,Y 473.828,Z 609.761,A -85,B 0,C 180,E1 14398.67,E2 14398.67} C_VEL
LIN {X 0,Y 475.356,Z 613.871,A -85,B 0,C 180,E1 14394.69,E2 14394.69} C_VEL
LIN {X 0,Y 476.494,Z 615.232,A -85,B 0,C 180,E1 14393.251,E2 14393.251} C_VEL
LIN {X 0,Y 479.687,Z 620.604,A -85,B 0,C 180,E1 14390.158,E2 14390.158} C_VEL
LIN {X 0,Y 482.487,Z 625.269,A -85,B 0,C 180,E1 14388.1,E2 14388.1} C_VEL
LIN {X 0,Y 485.044,Z 629.568,A -85,B 0,C 180,E1 14386.499,E2 14386.499} C_VEL
LIN {X 0,Y 490.203,Z 639.728,A -85,B 0,C 180,E1 14383.693,E2 14383.693} C_VEL
LIN {X 0,Y 471.589,Z 852.841,A -85,B 0,C 180,E1 14380.446,E2 14380.446} C_VEL
LIN {X 0,Y 467.225,Z 899.992,A -85,B 0,C 180,E1 14379.704,E2 14379.704} C_VEL
LIN {X 0,Y 462.826,Z 928.44,A -85,B 0,C 180,E1 14379.167,E2 14379.167} C_VEL
LIN {X 0,Y 458.247,Z 950.746,A -85,B 0,C 180,E1 14378.65,E2 14378.65} C_VEL
LIN {X 0,Y 453.088,Z 971.807,A -85,B 0,C 180,E1 14378.043,E2 14378.043} C_VEL
LIN {X 0,Y 447.08,Z 992.918,A -85,B 0,C 180,E1 14377.309,E2 14377.309} C_VEL
LIN {X 0,Y 438.609,Z 1018.858,A -85,B 0,C 180,E1 14376.202,E2 14376.202} C_VEL
LIN {X 0,Y 429.675,Z 1042.361,A -85,B 0,C 180,E1 14374.968,E2 14374.968} C_VEL
LIN {X 0,Y 421.834,Z 1061.169,A -85,B 0,C 180,E1 14373.796,E2 14373.796} C_VEL
LIN {X 0,Y 413.336,Z 1079.843,A -85,B 0,C 180,E1 14372.455,E2 14372.455} C_VEL
LIN {X 0,Y 403.632,Z 1099.65,A -85,B 0,C 180,E1 14370.79,E2 14370.79} C_VEL
LIN {X 0,Y 390.98,Z 1123.371,A -85,B 0,C 180,E1 14368.395,E2 14368.395} C_VEL
LIN {X 0,Y 381.046,Z 1140.749,A -85,B 0,C 180,E1 14366.294,E2 14366.294} C_VEL
LIN {X 0,Y 371.641,Z 1156.473,A -85,B 0,C 180,E1 14364.087,E2 14364.087} C_VEL
LIN {X 0,Y 362.125,Z 1171.81,A -85,B 0,C 180,E1 14361.591,E2 14361.591} C_VEL
LIN {X 0,Y 350.589,Z 1189.865,A -85,B 0,C 180,E1 14358.113,E2 14358.113} C_VEL
LIN {X 0,Y 341.057,Z 1204.414,A -85,B 0,C 180,E1 14354.725,E2 14354.725} C_VEL
LIN {X 0,Y 333.386,Z 1216.187,A -85,B 0,C 180,E1 14351.523,E2 14351.523} C_VEL
LIN {X 0,Y 326.341,Z 1227.244,A -85,B 0,C 180,E1 14348.021,E2 14348.021} C_VEL
LIN {X 0,Y 318.996,Z 1239.379,A -85,B 0,C 180,E1 14343.489,E2 14343.489} C_VEL
LIN {X 0,Y 313.27,Z 1249.461,A -85,B 0,C 180,E1 14338.821,E2 14338.821} C_VEL
LIN {X 0,Y 309.531,Z 1256.986,A -85,B 0,C 180,E1 14334.635,E2 14334.635} C_VEL
LIN {X 0,Y 306.973,Z 1263.001,A -85,B 0,C 180,E1 14330.604,E2 14330.604} C_VEL
LIN {X 0,Y 305.325,Z 1267.912,A -85,B 0,C 180,E1 14326.561,E2 14326.561} C_VEL
LIN {X 0,Y 304.332,Z 1272.241,A -85,B 0,C 180,E1 14321.954,E2 14321.954} C_VEL
LIN {X 0,Y 304.003,Z 1275.317,A -85,B 0,C 180,E1 14316.998,E2 14316.998} C_VEL
LIN {X 0,Y 303.978,Z 1276.644,A -85,B 0,C 180,E1 14312.837,E2 14312.837} C_VEL
LIN {X 0,Y 303.959,Z 1276.859,A -85,B 0,C 180,E1 14308.878,E2 14308.878} C_VEL
LIN {X 0,Y 303.975,Z 1276.104,A -85,B 0,C 180,E1 14305.103,E2 14305.103} C_VEL
LIN {X 0,Y 304.058,Z 1274.283,A -85,B 0,C 180,E1 14301.118,E2 14301.118} C_VEL
LIN {X 0,Y 304.448,Z 1271.561,A -85,B 0,C 180,E1 14297.274,E2 14297.274} C_VEL
LIN {X 0,Y 305.385,Z 1267.704,A -85,B 0,C 180,E1 14293.264,E2 14293.264} C_VEL
LIN {X 0,Y 307.069,Z 1262.746,A -85,B 0,C 180,E1 14289.221,E2 14289.221} C_VEL
LIN {X 0,Y 309.713,Z 1256.563,A -85,B 0,C 180,E1 14285.121,E2 14285.121} C_VEL
LIN {X 0,Y 314.064,Z 1248.01,A -85,B 0,C 180,E1 14280.442,E2 14280.442} C_VEL
LIN {X 0,Y 320.294,Z 1237.042,A -85,B 0,C 180,E1 14275.607,E2 14275.607} C_VEL
LIN {X 0,Y 326.637,Z 1226.728,A -85,B 0,C 180,E1 14271.817,E2 14271.817} C_VEL
LIN {X 0,Y 333.345,Z 1216.193,A -85,B 0,C 180,E1 14268.492,E2 14268.492} C_VEL
LIN {X 0,Y 341.437,Z 1203.766,A -85,B 0,C 180,E1 14265.123,E2 14265.123} C_VEL
LIN {X 0,Y 351.994,Z 1187.644,A -85,B 0,C 180,E1 14261.431,E2 14261.431} C_VEL
LIN {X 0,Y 362.19,Z 1171.59,A -85,B 0,C 180,E1 14258.385,E2 14258.385} C_VEL
LIN {X 0,Y 371.617,Z 1156.385,A -85,B 0,C 180,E1 14255.914,E2 14255.914} C_VEL
LIN {X 0,Y 380.976,Z 1140.72,A -85,B 0,C 180,E1 14253.715,E2 14253.715} C_VEL
LIN {X 0,Y 391.225,Z 1122.769,A -85,B 0,C 180,E1 14251.549,E2 14251.549} C_VEL
LIN {X 0,Y 403.554,Z 1099.583,A -85,B 0,C 180,E1 14249.216,E2 14249.216} C_VEL
LIN {X 0,Y 413.253,Z 1079.765,A -85,B 0,C 180,E1 14247.55,E2 14247.55} C_VEL
LIN {X 0,Y 421.749,Z 1061.081,A -85,B 0,C 180,E1 14246.208,E2 14246.208} C_VEL
LIN {X 0,Y 430.077,Z 1041.064,A -85,B 0,C 180,E1 14244.967,E2 14244.967} C_VEL
LIN {X 0,Y 439.768,Z 1015.12,A -85,B 0,C 180,E1 14243.633,E2 14243.633} C_VEL
LIN {X 0,Y 446.989,Z 992.761,A -85,B 0,C 180,E1 14242.694,E2 14242.694} C_VEL
LIN {X 0,Y 452.997,Z 971.619,A -85,B 0,C 180,E1 14241.959,E2 14241.959} C_VEL
LIN {X 0,Y 458.231,Z 950.18,A -85,B 0,C 180,E1 14241.343,E2 14241.343} C_VEL
LIN {X 0,Y 462.959,Z 926.985,A -85,B 0,C 180,E1 14240.81,E2 14240.81} C_VEL
LIN {X 0,Y 467.411,Z 896.787,A -85,B 0,C 180,E1 14240.25,E2 14240.25} C_VEL
LIN {X 0,Y 473.125,Z 832.988,A -85,B 0,C 180,E1 14239.257,E2 14239.257} C_VEL
LIN {X 0,Y 490.032,Z 639.636,A -85,B 0,C 180,E1 14236.309,E2 14236.309} C_VEL
LIN {X 0,Y 484.629,Z 628.953,A -85,B 0,C 180,E1 14233.361,E2 14233.361} C_VEL
LIN {X 0,Y 480.785,Z 622.642,A -85,B 0,C 180,E1 14230.849,E2 14230.849} C_VEL
LIN {X 0,Y 478.633,Z 619.105,A -85,B 0,C 180,E1 14229.135,E2 14229.135} C_VEL
LIN {X 0,Y 475.972,Z 614.613,A -85,B 0,C 180,E1 14226.393,E2 14226.393} C_VEL
LIN {X 0,Y 473.786,Z 610.954,A -85,B 0,C 180,E1 14222.54,E2 14222.54} C_VEL
LIN {X 0,Y 473.548,Z 609.564,A -85,B 0,C 180,E1 14221.21,E2 14221.21} C_VEL
LIN {X 0,Y 473.611,Z 609.702,A -85,B 0,C 180,E1 14217.943,E2 14217.943} C_VEL
LIN {X 0,Y 475.108,Z 613.705,A -85,B 0,C 180,E1 14214.202,E2 14214.202} C_VEL
LIN {X 0,Y 476.302,Z 615.148,A -85,B 0,C 180,E1 14212.703,E2 14212.703} C_VEL
LIN {X 0,Y 479.387,Z 620.296,A -85,B 0,C 180,E1 14209.727,E2 14209.727} C_VEL
LIN {X 0,Y 482.445,Z 625.382,A -85,B 0,C 180,E1 14207.492,E2 14207.492} C_VEL
LIN {X 0,Y 486.334,Z 631.682,A -85,B 0,C 180,E1 14205.169,E2 14205.169} C_VEL
LIN {X 0,Y 489.941,Z 638.071,A -85,B 0,C 180,E1 14203.299,E2 14203.299} C_VEL
LIN {X 0,Y 470.84,Z 856.175,A -85,B 0,C 180,E1 14199.986,E2 14199.986} C_VEL
LIN {X 0,Y 467.104,Z 893.655,A -85,B 0,C 180,E1 14199.384,E2 14199.384} C_VEL
LIN {X 0,Y 463.053,Z 918.958,A -85,B 0,C 180,E1 14198.878,E2 14198.878} C_VEL
LIN {X 0,Y 458.729,Z 940.38,A -85,B 0,C 180,E1 14198.334,E2 14198.334} C_VEL
LIN {X 0,Y 453.621,Z 961.489,A -85,B 0,C 180,E1 14197.679,E2 14197.679} C_VEL
LIN {X 0,Y 447.024,Z 984.826,A -85,B 0,C 180,E1 14196.803,E2 14196.803} C_VEL
LIN {X 0,Y 438.468,Z 1010.441,A -85,B 0,C 180,E1 14195.622,E2 14195.622} C_VEL
LIN {X 0,Y 430.837,Z 1030.562,A -85,B 0,C 180,E1 14194.506,E2 14194.506} C_VEL
LIN {X 0,Y 422.991,Z 1049.304,A -85,B 0,C 180,E1 14193.301,E2 14193.301} C_VEL
LIN {X 0,Y 414.656,Z 1067.603,A -85,B 0,C 180,E1 14191.933,E2 14191.933} C_VEL
LIN {X 0,Y 405.457,Z 1086.24,A -85,B 0,C 180,E1 14190.324,E2 14190.324} C_VEL
LIN {X 0,Y 393.216,Z 1109.03,A -85,B 0,C 180,E1 14187.981,E2 14187.981} C_VEL
LIN {X 0,Y 383.287,Z 1126.128,A -85,B 0,C 180,E1 14185.883,E2 14185.883} C_VEL
LIN {X 0,Y 374.229,Z 1140.954,A -85,B 0,C 180,E1 14183.778,E2 14183.778} C_VEL
LIN {X 0,Y 364.819,Z 1155.737,A -85,B 0,C 180,E1 14181.348,E2 14181.348} C_VEL
LIN {X 0,Y 354.089,Z 1172.111,A -85,B 0,C 180,E1 14178.187,E2 14178.187} C_VEL
LIN {X 0,Y 343.286,Z 1187.938,A -85,B 0,C 180,E1 14174.47,E2 14174.47} C_VEL
LIN {X 0,Y 335.266,Z 1199.611,A -85,B 0,C 180,E1 14171.218,E2 14171.218} C_VEL
LIN {X 0,Y 328.046,Z 1210.201,A -85,B 0,C 180,E1 14167.769,E2 14167.769} C_VEL
LIN {X 0,Y 320.785,Z 1221.324,A -85,B 0,C 180,E1 14163.472,E2 14163.472} C_VEL
LIN {X 0,Y 314.509,Z 1231.35,A -85,B 0,C 180,E1 14158.662,E2 14158.662} C_VEL
LIN {X 0,Y 310.544,Z 1238.417,A -85,B 0,C 180,E1 14154.531,E2 14154.531} C_VEL
LIN {X 0,Y 307.748,Z 1244.061,A -85,B 0,C 180,E1 14150.532,E2 14150.532} C_VEL
LIN {X 0,Y 305.865,Z 1248.64,A -85,B 0,C 180,E1 14146.514,E2 14146.514} C_VEL
LIN {X 0,Y 304.695,Z 1252.498,A -85,B 0,C 180,E1 14142.114,E2 14142.114} C_VEL
LIN {X 0,Y 304.135,Z 1255.426,A -85,B 0,C 180,E1 14137.168,E2 14137.168} C_VEL
LIN {X 0,Y 303.998,Z 1256.709,A -85,B 0,C 180,E1 14132.819,E2 14132.819} C_VEL
LIN {X 0,Y 303.96,Z 1256.914,A -85,B 0,C 180,E1 14128.861,E2 14128.861} C_VEL
LIN {X 0,Y 304.032,Z 1256.235,A -85,B 0,C 180,E1 14125.086,E2 14125.086} C_VEL
LIN {X 0,Y 304.247,Z 1254.58,A -85,B 0,C 180,E1 14121.106,E2 14121.106} C_VEL
LIN {X 0,Y 304.828,Z 1251.954,A -85,B 0,C 180,E1 14117.104,E2 14117.104} C_VEL
LIN {X 0,Y 305.991,Z 1248.33,A -85,B 0,C 180,E1 14113.085,E2 14113.085} C_VEL
LIN {X 0,Y 307.941,Z 1243.678,A -85,B 0,C 180,E1 14109.066,E2 14109.066} C_VEL
LIN {X 0,Y 310.975,Z 1237.666,A -85,B 0,C 180,E1 14104.878,E2 14104.878} C_VEL
LIN {X 0,Y 315.993,Z 1229.049,A -85,B 0,C 180,E1 14099.995,E2 14099.995} C_VEL
LIN {X 0,Y 322.364,Z 1218.825,A -85,B 0,C 180,E1 14095.408,E2 14095.408} C_VEL
LIN {X 0,Y 328.625,Z 1209.397,A -85,B 0,C 180,E1 14091.847,E2 14091.847} C_VEL
LIN {X 0,Y 335.934,Z 1198.712,A -85,B 0,C 180,E1 14088.406,E2 14088.406} C_VEL
LIN {X 0,Y 345.56,Z 1184.805,A -85,B 0,C 180,E1 14084.61,E2 14084.61} C_VEL
LIN {X 0,Y 356.216,Z 1168.928,A -85,B 0,C 180,E1 14081.059,E2 14081.059} C_VEL
LIN {X 0,Y 365.459,Z 1154.868,A -85,B 0,C 180,E1 14078.394,E2 14078.394} C_VEL
LIN {X 0,Y 374.669,Z 1140.39,A -85,B 0,C 180,E1 14076.031,E2 14076.031} C_VEL
LIN {X 0,Y 385.321,Z 1122.925,A -85,B 0,C 180,E1 14073.587,E2 14073.587} C_VEL
LIN {X 0,Y 388.156,Z 1118.069,A -85,B 0,C 180,E1 14072.977,E2 14072.977} C_VEL
LIN {X 0,Y 390.594,Z 1112.867,A -85,B 0,C 180,E1 14072.221,E2 14072.221} C_VEL
LIN {X 0,Y 394.66,Z 1100.164,A -85,B 0,C 180,E1 14070.022,E2 14070.022} C_VEL
LIN {X 0,Y 397.271,Z 1094.572,A -85,B 0,C 180,E1 14069.328,E2 14069.328} C_VEL
LIN {X 0,Y 409.357,Z 1071.31,A -85,B 0,C 180,E1 14067.232,E2 14067.232} C_VEL
LIN {X 0,Y 418.558,Z 1051.751,A -85,B 0,C 180,E1 14065.754,E2 14065.754} C_VEL
LIN {X 0,Y 426.558,Z 1033.233,A -85,B 0,C 180,E1 14064.556,E2 14064.556} C_VEL
LIN {X 0,Y 434.026,Z 1014.18,A -85,B 0,C 180,E1 14063.488,E2 14063.488} C_VEL
LIN {X 0,Y 441.512,Z 992.921,A -85,B 0,C 180,E1 14062.475,E2 14062.475} C_VEL
LIN {X 0,Y 449.753,Z 965.682,A -85,B 0,C 180,E1 14061.407,E2 14061.407} C_VEL
LIN {X 0,Y 455.588,Z 942.4,A -85,B 0,C 180,E1 14060.68,E2 14060.68} C_VEL
LIN {X 0,Y 460.026,Z 921.101,A -85,B 0,C 180,E1 14060.135,E2 14060.135} C_VEL
LIN {X 0,Y 463.732,Z 899.006,A -85,B 0,C 180,E1 14059.686,E2 14059.686} C_VEL
LIN {X 0,Y 467.072,Z 870.813,A -85,B 0,C 180,E1 14059.216,E2 14059.216} C_VEL
LIN {X 0,Y 486.949,Z 648.521,A -85,B 0,C 180,E1 14055.857,E2 14055.857} C_VEL
LIN {X 0,Y 487.341,Z 643.482,A -85,B 0,C 180,E1 14055.752,E2 14055.752} C_VEL
LIN {X 0,Y 482.504,Z 635.142,A -85,B 0,C 180,E1 14052.994,E2 14052.994} C_VEL
LIN {X 0,Y 479.527,Z 630.241,A -85,B 0,C 180,E1 14050.938,E2 14050.938} C_VEL
LIN {X 0,Y 477.533,Z 626.821,A -85,B 0,C 180,E1 14049.278,E2 14049.278} C_VEL
LIN {X 0,Y 474.986,Z 622.443,A -85,B 0,C 180,E1 14046.527,E2 14046.527} C_VEL
LIN {X 0,Y 472.903,Z 618.475,A -85,B 0,C 180,E1 14042.302,E2 14042.302} C_VEL
LIN {X 0,Y 472.795,Z 617.527,A -85,B 0,C 180,E1 14041.333,E2 14041.333} C_VEL
LIN {X 0,Y 472.842,Z 617.789,A -85,B 0,C 180,E1 14038.667,E2 14038.667} C_VEL
LIN {X 0,Y 474.38,Z 621.851,A -85,B 0,C 180,E1 14034.679,E2 14034.679} C_VEL
LIN {X 0,Y 475.407,Z 623.156,A -85,B 0,C 180,E1 14033.357,E2 14033.357} C_VEL
LIN {X 0,Y 478.411,Z 628.292,A -85,B 0,C 180,E1 14030.375,E2 14030.375} C_VEL
LIN {X 0,Y 481.146,Z 632.966,A -85,B 0,C 180,E1 14028.31,E2 14028.31} C_VEL
LIN {X 0,Y 483.554,Z 637.133,A -85,B 0,C 180,E1 14026.761,E2 14026.761} C_VEL
LIN {X 0,Y 487.485,Z 645.143,A -85,B 0,C 180,E1 14024.515,E2 14024.515} C_VEL
LIN {X 0,Y 468.211,Z 861.126,A -85,B 0,C 180,E1 14021.243,E2 14021.243} C_VEL
LIN {X 0,Y 464.169,Z 902.56,A -85,B 0,C 180,E1 14020.588,E2 14020.588} C_VEL
LIN {X 0,Y 459.771,Z 929.495,A -85,B 0,C 180,E1 14020.077,E2 14020.077} C_VEL
LIN {X 0,Y 455.179,Z 951.323,A -85,B 0,C 180,E1 14019.575,E2 14019.575} C_VEL
LIN {X 0,Y 449.927,Z 972.294,A -85,B 0,C 180,E1 14018.976,E2 14018.976} C_VEL
LIN {X 0,Y 443.258,Z 995.154,A -85,B 0,C 180,E1 14018.183,E2 14018.183} C_VEL
LIN {X 0,Y 433.965,Z 1022.316,A -85,B 0,C 180,E1 14017.004,E2 14017.004} C_VEL
LIN {X 0,Y 426.021,Z 1042.708,A -85,B 0,C 180,E1 14015.931,E2 14015.931} C_VEL
LIN {X 0,Y 417.899,Z 1061.722,A -85,B 0,C 180,E1 14014.753,E2 14014.753} C_VEL
LIN {X 0,Y 408.872,Z 1081.06,A -85,B 0,C 180,E1 14013.365,E2 14013.365} C_VEL
LIN {X 0,Y 397.383,Z 1103.812,A -85,B 0,C 180,E1 14011.427,E2 14011.427} C_VEL
LIN {X 0,Y 385.728,Z 1124.729,A -85,B 0,C 180,E1 14009.262,E2 14009.262} C_VEL
LIN {X 0,Y 375.846,Z 1141.504,A -85,B 0,C 180,E1 14007.219,E2 14007.219} C_VEL
LIN {X 0,Y 365.901,Z 1157.609,A -85,B 0,C 180,E1 14004.936,E2 14004.936} C_VEL
LIN {X 0,Y 354.358,Z 1175.619,A -85,B 0,C 180,E1 14001.937,E2 14001.937} C_VEL
LIN {X 0,Y 343.031,Z 1192.443,A -85,B 0,C 180,E1 13998.522,E2 13998.522} C_VEL
LIN {X 0,Y 334.215,Z 1205.433,A -85,B 0,C 180,E1 13995.409,E2 13995.409} C_VEL
LIN {X 0,Y 326.24,Z 1217.194,A -85,B 0,C 180,E1 13992.123,E2 13992.123} C_VEL
LIN {X 0,Y 317.567,Z 1230.355,A -85,B 0,C 180,E1 13987.786,E2 13987.786} C_VEL
LIN {X 0,Y 310.131,Z 1242.026,A -85,B 0,C 180,E1 13983.024,E2 13983.024} C_VEL
LIN {X 0,Y 305.327,Z 1250.278,A -85,B 0,C 180,E1 13978.999,E2 13978.999} C_VEL
LIN {X 0,Y 301.665,Z 1257.338,A -85,B 0,C 180,E1 13974.903,E2 13974.903} C_VEL
LIN {X 0,Y 298.818,Z 1263.782,A -85,B 0,C 180,E1 13970.373,E2 13970.373} C_VEL
LIN {X 0,Y 296.884,Z 1269.644,A -85,B 0,C 180,E1 13965.039,E2 13965.039} C_VEL
LIN {X 0,Y 296.16,Z 1273.182,A -85,B 0,C 180,E1 13960.513,E2 13960.513} C_VEL
LIN {X 0,Y 295.997,Z 1275.34,A -85,B 0,C 180,E1 13956.409,E2 13956.409} C_VEL
LIN {X 0,Y 295.983,Z 1276.43,A -85,B 0,C 180,E1 13952.526,E2 13952.526} C_VEL
LIN {X 0,Y 295.964,Z 1276.596,A -85,B 0,C 180,E1 13948.847,E2 13948.847} C_VEL
LIN {X 0,Y 295.978,Z 1275.84,A -85,B 0,C 180,E1 13944.97,E2 13944.97} C_VEL
LIN {X 0,Y 296.063,Z 1274.017,A -85,B 0,C 180,E1 13940.876,E2 13940.876} C_VEL
LIN {X 0,Y 296.494,Z 1271.314,A -85,B 0,C 180,E1 13936.951,E2 13936.951} C_VEL
LIN {X 0,Y 297.525,Z 1267.434,A -85,B 0,C 180,E1 13932.808,E2 13932.808} C_VEL
LIN {X 0,Y 299.333,Z 1262.473,A -85,B 0,C 180,E1 13928.658,E2 13928.658} C_VEL
LIN {X 0,Y 302.099,Z 1256.403,A -85,B 0,C 180,E1 13924.526,E2 13924.526} C_VEL
LIN {X 0,Y 306.352,Z 1248.461,A -85,B 0,C 180,E1 13920.053,E2 13920.053} C_VEL
LIN {X 0,Y 313.376,Z 1236.764,A -85,B 0,C 180,E1 13914.736,E2 13914.736} C_VEL
LIN {X 0,Y 320.033,Z 1226.448,A -85,B 0,C 180,E1 13910.881,E2 13910.881} C_VEL
LIN {X 0,Y 327.246,Z 1215.626,A -85,B 0,C 180,E1 13907.423,E2 13907.423} C_VEL
LIN {X 0,Y 335.496,Z 1203.487,A -85,B 0,C 180,E1 13904.104,E2 13904.104} C_VEL
LIN {X 0,Y 346.47,Z 1187.365,A -85,B 0,C 180,E1 13900.385,E2 13900.385} C_VEL
LIN {X 0,Y 357.029,Z 1171.312,A -85,B 0,C 180,E1 13897.327,E2 13897.327} C_VEL
LIN {X 0,Y 366.719,Z 1156.173,A -85,B 0,C 180,E1 13894.862,E2 13894.862} C_VEL
LIN {X 0,Y 376.4,Z 1140.443,A -85,B 0,C 180,E1 13892.656,E2 13892.656} C_VEL
LIN {X 0,Y 386.932,Z 1122.493,A -85,B 0,C 180,E1 13890.498,E2 13890.498} C_VEL
LIN {X 0,Y 399.734,Z 1098.995,A -85,B 0,C 180,E1 13888.152,E2 13888.152} C_VEL
LIN {X 0,Y 409.324,Z 1079.853,A -85,B 0,C 180,E1 13886.553,E2 13886.553} C_VEL
LIN {X 0,Y 418.26,Z 1060.623,A -85,B 0,C 180,E1 13885.184,E2 13885.184} C_VEL
LIN {X 0,Y 426.684,Z 1040.79,A -85,B 0,C 180,E1 13883.969,E2 13883.969} C_VEL
LIN {X 0,Y 436.563,Z 1014.845,A -85,B 0,C 180,E1 13882.652,E2 13882.652} C_VEL
LIN {X 0,Y 443.921,Z 992.487,A -85,B 0,C 180,E1 13881.727,E2 13881.727} C_VEL
LIN {X 0,Y 450.033,Z 971.344,A -85,B 0,C 180,E1 13881.003,E2 13881.003} C_VEL
LIN {X 0,Y 455.304,Z 950.127,A -85,B 0,C 180,E1 13880.402,E2 13880.402} C_VEL
LIN {X 0,Y 460.058,Z 927.231,A -85,B 0,C 180,E1 13879.884,E2 13879.884} C_VEL
LIN {X 0,Y 464.673,Z 896.609,A -85,B 0,C 180,E1 13879.32,E2 13879.32} C_VEL
LIN {X 0,Y 470.434,Z 833.781,A -85,B 0,C 180,E1 13878.347,E2 13878.347} C_VEL
LIN {X 0,Y 487.316,Z 644.967,A -85,B 0,C 180,E1 13875.486,E2 13875.486} C_VEL
LIN {X 0,Y 482.583,Z 635.475,A -85,B 0,C 180,E1 13872.748,E2 13872.748} C_VEL
LIN {X 0,Y 479.239,Z 629.964,A -85,B 0,C 180,E1 13870.458,E2 13870.458} C_VEL
LIN {X 0,Y 477.375,Z 626.822,A -85,B 0,C 180,E1 13868.917,E2 13868.917} C_VEL
LIN {X 0,Y 474.793,Z 622.404,A -85,B 0,C 180,E1 13866.166,E2 13866.166} C_VEL
LIN {X 0,Y 472.744,Z 618.681,A -85,B 0,C 180,E1 13862.303,E2 13862.303} C_VEL
LIN {X 0,Y 472.573,Z 617.505,A -85,B 0,C 180,E1 13861.212,E2 13861.212} C_VEL
LIN {X 0,Y 472.623,Z 617.752,A -85,B 0,C 180,E1 13857.939,E2 13857.939} C_VEL
LIN {X 0,Y 474.305,Z 621.893,A -85,B 0,C 180,E1 13853.949,E2 13853.949} C_VEL
LIN {X 0,Y 475.215,Z 623.074,A -85,B 0,C 180,E1 13852.808,E2 13852.808} C_VEL
LIN {X 0,Y 478.182,Z 628.126,A -85,B 0,C 180,E1 13849.884,E2 13849.884} C_VEL
LIN {X 0,Y 481.101,Z 633.08,A -85,B 0,C 180,E1 13847.7,E2 13847.7} C_VEL
LIN {X 0,Y 484.814,Z 639.227,A -85,B 0,C 180,E1 13845.427,E2 13845.427} C_VEL
LIN {X 0,Y 487.208,Z 643.735,A -85,B 0,C 180,E1 13844.119,E2 13844.119} C_VEL
LIN {X 0,Y 467.453,Z 864.598,A -85,B 0,C 180,E1 13840.782,E2 13840.782} C_VEL
LIN {X 0,Y 463.781,Z 897.658,A -85,B 0,C 180,E1 13840.241,E2 13840.241} C_VEL
LIN {X 0,Y 460,Z 920.43,A -85,B 0,C 180,E1 13839.782,E2 13839.782} C_VEL
LIN {X 0,Y 455.583,Z 941.734,A -85,B 0,C 180,E1 13839.241,E2 13839.241} C_VEL
LIN {X 0,Y 450.242,Z 963.235,A -85,B 0,C 180,E1 13838.576,E2 13838.576} C_VEL
LIN {X 0,Y 442.772,Z 988.799,A -85,B 0,C 180,E1 13837.607,E2 13837.607} C_VEL
LIN {X 0,Y 434.448,Z 1012.684,A -85,B 0,C 180,E1 13836.491,E2 13836.491} C_VEL
LIN {X 0,Y 427.039,Z 1031.727,A -85,B 0,C 180,E1 13835.435,E2 13835.435} C_VEL
LIN {X 0,Y 419.074,Z 1050.3,A -85,B 0,C 180,E1 13834.244,E2 13834.244} C_VEL
LIN {X 0,Y 410.529,Z 1068.603,A -85,B 0,C 180,E1 13832.88,E2 13832.88} C_VEL
LIN {X 0,Y 400.194,Z 1089.001,A -85,B 0,C 180,E1 13831.112,E2 13831.112} C_VEL
LIN {X 0,Y 388.286,Z 1110.367,A -85,B 0,C 180,E1 13828.886,E2 13828.886} C_VEL
LIN {X 0,Y 378.314,Z 1127.053,A -85,B 0,C 180,E1 13826.831,E2 13826.831} C_VEL
LIN {X 0,Y 368.808,Z 1142.142,A -85,B 0,C 180,E1 13824.675,E2 13824.675} C_VEL
LIN {X 0,Y 359.108,Z 1156.893,A -85,B 0,C 180,E1 13822.225,E2 13822.225} C_VEL
LIN {X 0,Y 347.59,Z 1173.847,A -85,B 0,C 180,E1 13818.895,E2 13818.895} C_VEL
LIN {X 0,Y 336.975,Z 1188.782,A -85,B 0,C 180,E1 13815.312,E2 13815.312} C_VEL
LIN {X 0,Y 328.895,Z 1200.086,A -85,B 0,C 180,E1 13812.115,E2 13812.115} C_VEL
LIN {X 0,Y 321.496,Z 1210.477,A -85,B 0,C 180,E1 13808.679,E2 13808.679} C_VEL
LIN {X 0,Y 313.59,Z 1222.044,A -85,B 0,C 180,E1 13804.125,E2 13804.125} C_VEL
LIN {X 0,Y 307.047,Z 1231.94,A -85,B 0,C 180,E1 13799.228,E2 13799.228} C_VEL
LIN {X 0,Y 303.042,Z 1238.689,A -85,B 0,C 180,E1 13795.18,E2 13795.18} C_VEL
LIN {X 0,Y 300.059,Z 1244.332,A -85,B 0,C 180,E1 13791.083,E2 13791.083} C_VEL
LIN {X 0,Y 298.043,Z 1248.908,A -85,B 0,C 180,E1 13786.96,E2 13786.96} C_VEL
LIN {X 0,Y 296.729,Z 1252.918,A -85,B 0,C 180,E1 13782.247,E2 13782.247} C_VEL
LIN {X 0,Y 296.141,Z 1255.755,A -85,B 0,C 180,E1 13777.167,E2 13777.167} C_VEL
LIN {X 0,Y 296,Z 1256.993,A -85,B 0,C 180,E1 13772.702,E2 13772.702} C_VEL
LIN {X 0,Y 295.966,Z 1257.176,A -85,B 0,C 180,E1 13768.83,E2 13768.83} C_VEL
LIN {X 0,Y 296.04,Z 1256.498,A -85,B 0,C 180,E1 13764.953,E2 13764.953} C_VEL
LIN {X 0,Y 296.282,Z 1254.844,A -85,B 0,C 180,E1 13760.865,E2 13760.865} C_VEL
LIN {X 0,Y 296.922,Z 1252.185,A -85,B 0,C 180,E1 13756.71,E2 13756.71} C_VEL
LIN {X 0,Y 298.181,Z 1248.598,A -85,B 0,C 180,E1 13752.628,E2 13752.628} C_VEL
LIN {X 0,Y 300.27,Z 1243.947,A -85,B 0,C 180,E1 13748.505,E2 13748.505} C_VEL
LIN {X 0,Y 303.5,Z 1237.936,A -85,B 0,C 180,E1 13744.215,E2 13744.215} C_VEL
LIN {X 0,Y 308.813,Z 1229.321,A -85,B 0,C 180,E1 13739.223,E2 13739.223} C_VEL
LIN {X 0,Y 315.583,Z 1219.02,A -85,B 0,C 180,E1 13734.516,E2 13734.516} C_VEL
LIN {X 0,Y 322.47,Z 1209.166,A -85,B 0,C 180,E1 13730.754,E2 13730.754} C_VEL
LIN {X 0,Y 330.547,Z 1197.862,A -85,B 0,C 180,E1 13727.101,E2 13727.101} C_VEL
LIN {X 0,Y 342.082,Z 1181.683,A -85,B 0,C 180,E1 13722.798,E2 13722.798} C_VEL
LIN {X 0,Y 351.709,Z 1167.877,A -85,B 0,C 180,E1 13719.767,E2 13719.767} C_VEL
LIN {X 0,Y 360.676,Z 1154.665,A -85,B 0,C 180,E1 13717.277,E2 13717.277} C_VEL
LIN {X 0,Y 371.041,Z 1138.833,A -85,B 0,C 180,E1 13714.715,E2 13714.715} C_VEL
LIN {X 0,Y 383.966,Z 1117.93,A -85,B 0,C 180,E1 13711.896,E2 13711.896} C_VEL
LIN {X 0,Y 394.34,Z 1099.826,A -85,B 0,C 180,E1 13709.861,E2 13709.861} C_VEL
LIN {X 0,Y 397.271,Z 1094.572,A -85,B 0,C 180,E1 13709.328,E2 13709.328} C_VEL
LIN {X 0,Y 399.891,Z 1088.99,A -85,B 0,C 180,E1 13708.651,E2 13708.651} C_VEL
LIN {X 0,Y 404.586,Z 1074.514,A -85,B 0,C 180,E1 13706.541,E2 13706.541} C_VEL
LIN {X 0,Y 406.768,Z 1069.37,A -85,B 0,C 180,E1 13706.033,E2 13706.033} C_VEL
LIN {X 0,Y 415.454,Z 1051.208,A -85,B 0,C 180,E1 13704.687,E2 13704.687} C_VEL
LIN {X 0,Y 423.522,Z 1032.832,A -85,B 0,C 180,E1 13703.515,E2 13703.515} C_VEL
LIN {X 0,Y 431.281,Z 1013.347,A -85,B 0,C 180,E1 13702.444,E2 13702.444} C_VEL
LIN {X 0,Y 440.051,Z 988.685,A -85,B 0,C 180,E1 13701.305,E2 13701.305} C_VEL
LIN {X 0,Y 447.645,Z 963.065,A -85,B 0,C 180,E1 13700.352,E2 13700.352} C_VEL
LIN {X 0,Y 453.052,Z 941.604,A -85,B 0,C 180,E1 13699.7,E2 13699.7} C_VEL
LIN {X 0,Y 457.528,Z 920.311,A -85,B 0,C 180,E1 13699.169,E2 13699.169} C_VEL
LIN {X 0,Y 461.47,Z 896.831,A -85,B 0,C 180,E1 13698.705,E2 13698.705} C_VEL
LIN {X 0,Y 465.389,Z 861.038,A -85,B 0,C 180,E1 13698.131,E2 13698.131} C_VEL
LIN {X 0,Y 484.758,Z 649.315,A -85,B 0,C 180,E1 13694.95,E2 13694.95} C_VEL
LIN {X 0,Y 480.691,Z 642.129,A -85,B 0,C 180,E1 13692.494,E2 13692.494} C_VEL
LIN {X 0,Y 478.154,Z 637.81,A -85,B 0,C 180,E1 13690.665,E2 13690.665} C_VEL
LIN {X 0,Y 476.286,Z 634.538,A -85,B 0,C 180,E1 13689.059,E2 13689.059} C_VEL
LIN {X 0,Y 473.915,Z 630.326,A -85,B 0,C 180,E1 13686.42,E2 13686.42} C_VEL
LIN {X 0,Y 471.901,Z 626.354,A -85,B 0,C 180,E1 13682.186,E2 13682.186} C_VEL
LIN {X 0,Y 471.801,Z 625.467,A -85,B 0,C 180,E1 13681.214,E2 13681.214} C_VEL
LIN {X 0,Y 471.849,Z 625.668,A -85,B 0,C 180,E1 13678.786,E2 13678.786} C_VEL
LIN {X 0,Y 473.322,Z 629.731,A -85,B 0,C 180,E1 13674.788,E2 13674.788} C_VEL
LIN {X 0,Y 474.278,Z 630.962,A -85,B 0,C 180,E1 13673.524,E2 13673.524} C_VEL
LIN {X 0,Y 477.21,Z 636.115,A -85,B 0,C 180,E1 13670.533,E2 13670.533} C_VEL
LIN {X 0,Y 479.895,Z 640.813,A -85,B 0,C 180,E1 13668.462,E2 13668.462} C_VEL
LIN {X 0,Y 482.073,Z 644.696,A -85,B 0,C 180,E1 13667.025,E2 13667.025} C_VEL
LIN {X 0,Y 484.848,Z 650.757,A -85,B 0,C 180,E1 13665.345,E2 13665.345} C_VEL
LIN {X 0,Y 465.137,Z 867.025,A -85,B 0,C 180,E1 13662.089,E2 13662.089} C_VEL
LIN {X 0,Y 461.256,Z 904.265,A -85,B 0,C 180,E1 13661.496,E2 13661.496} C_VEL
LIN {X 0,Y 457.012,Z 929.635,A -85,B 0,C 180,E1 13661.018,E2 13661.018} C_VEL
LIN {X 0,Y 452.346,Z 951.408,A -85,B 0,C 180,E1 13660.524,E2 13660.524} C_VEL
LIN {X 0,Y 446.886,Z 972.78,A -85,B 0,C 180,E1 13659.921,E2 13659.921} C_VEL
LIN {X 0,Y 439.347,Z 998.034,A -85,B 0,C 180,E1 13659.046,E2 13659.046} C_VEL
LIN {X 0,Y 430.453,Z 1023.065,A -85,B 0,C 180,E1 13657.953,E2 13657.953} C_VEL
LIN {X 0,Y 422.543,Z 1042.927,A -85,B 0,C 180,E1 13656.917,E2 13656.917} C_VEL
LIN {X 0,Y 414.455,Z 1061.456,A -85,B 0,C 180,E1 13655.783,E2 13655.783} C_VEL
LIN {X 0,Y 405.342,Z 1080.58,A -85,B 0,C 180,E1 13654.425,E2 13654.425} C_VEL
LIN {X 0,Y 393.754,Z 1103.06,A -85,B 0,C 180,E1 13652.534,E2 13652.534} C_VEL
LIN {X 0,Y 381.839,Z 1123.954,A -85,B 0,C 180,E1 13650.395,E2 13650.395} C_VEL
LIN {X 0,Y 371.64,Z 1140.829,A -85,B 0,C 180,E1 13648.356,E2 13648.356} C_VEL
LIN {X 0,Y 362.059,Z 1155.928,A -85,B 0,C 180,E1 13646.237,E2 13646.237} C_VEL
LIN {X 0,Y 352.054,Z 1171.06,A -85,B 0,C 180,E1 13643.774,E2 13643.774} C_VEL
LIN {X 0,Y 339.861,Z 1188.9,A -85,B 0,C 180,E1 13640.325,E2 13640.325} C_VEL
LIN {X 0,Y 329.254,Z 1203.863,A -85,B 0,C 180,E1 13636.797,E2 13636.797} C_VEL
LIN {X 0,Y 320.907,Z 1215.634,A -85,B 0,C 180,E1 13633.527,E2 13633.527} C_VEL
LIN {X 0,Y 313.192,Z 1226.692,A -85,B 0,C 180,E1 13629.927,E2 13629.927} C_VEL
LIN {X 0,Y 305.073,Z 1238.828,A -85,B 0,C 180,E1 13625.237,E2 13625.237} C_VEL
LIN {X 0,Y 298.456,Z 1249.276,A -85,B 0,C 180,E1 13620.176,E2 13620.176} C_VEL
LIN {X 0,Y 294.43,Z 1256.439,A -85,B 0,C 180,E1 13615.99,E2 13615.99} C_VEL
LIN {X 0,Y 291.513,Z 1262.459,A -85,B 0,C 180,E1 13611.751,E2 13611.751} C_VEL
LIN {X 0,Y 289.541,Z 1267.588,A -85,B 0,C 180,E1 13607.285,E2 13607.285} C_VEL
LIN {X 0,Y 288.31,Z 1272.32,A -85,B 0,C 180,E1 13601.816,E2 13601.816} C_VEL
LIN {X 0,Y 288.008,Z 1274.932,A -85,B 0,C 180,E1 13596.988,E2 13596.988} C_VEL
LIN {X 0,Y 287.986,Z 1276.143,A -85,B 0,C 180,E1 13592.795,E2 13592.795} C_VEL
LIN {X 0,Y 287.969,Z 1276.334,A -85,B 0,C 180,E1 13588.815,E2 13588.815} C_VEL
LIN {X 0,Y 287.981,Z 1275.577,A -85,B 0,C 180,E1 13584.83,E2 13584.83} C_VEL
LIN {X 0,Y 288.065,Z 1273.87,A -85,B 0,C 180,E1 13580.822,E2 13580.822} C_VEL
LIN {X 0,Y 288.551,Z 1271.045,A -85,B 0,C 180,E1 13576.585,E2 13576.585} C_VEL
LIN {X 0,Y 289.675,Z 1267.14,A -85,B 0,C 180,E1 13572.306,E2 13572.306} C_VEL
LIN {X 0,Y 291.611,Z 1262.199,A -85,B 0,C 180,E1 13568.064,E2 13568.064} C_VEL
LIN {X 0,Y 294.577,Z 1256.128,A -85,B 0,C 180,E1 13563.827,E2 13563.827} C_VEL
LIN {X 0,Y 299.156,Z 1248.099,A -85,B 0,C 180,E1 13559.204,E2 13559.204} C_VEL
LIN {X 0,Y 306.53,Z 1236.486,A -85,B 0,C 180,E1 13553.827,E2 13553.827} C_VEL
LIN {X 0,Y 313.51,Z 1226.169,A -85,B 0,C 180,E1 13549.905,E2 13549.905} C_VEL
LIN {X 0,Y 320.863,Z 1215.634,A -85,B 0,C 180,E1 13546.488,E2 13546.488} C_VEL
LIN {X 0,Y 329.671,Z 1203.208,A -85,B 0,C 180,E1 13543.049,E2 13543.049} C_VEL
LIN {X 0,Y 341.163,Z 1186.941,A -85,B 0,C 180,E1 13539.276,E2 13539.276} C_VEL
LIN {X 0,Y 352.557,Z 1170.174,A -85,B 0,C 180,E1 13536.088,E2 13536.088} C_VEL
LIN {X 0,Y 362.372,Z 1155.306,A -85,B 0,C 180,E1 13533.685,E2 13533.685} C_VEL
LIN {X 0,Y 372.35,Z 1139.539,A -85,B 0,C 180,E1 13531.491,E2 13531.491} C_VEL
LIN {X 0,Y 384.634,Z 1119.149,A -85,B 0,C 180,E1 13529.086,E2 13529.086} C_VEL
LIN {X 0,Y 396.489,Z 1097.588,A -85,B 0,C 180,E1 13526.997,E2 13526.997} C_VEL
LIN {X 0,Y 405.895,Z 1079.182,A -85,B 0,C 180,E1 13525.48,E2 13525.48} C_VEL
LIN {X 0,Y 414.703,Z 1060.613,A -85,B 0,C 180,E1 13524.173,E2 13524.173} C_VEL
LIN {X 0,Y 423.424,Z 1040.516,A -85,B 0,C 180,E1 13522.957,E2 13522.957} C_VEL
LIN {X 0,Y 433.49,Z 1014.565,A -85,B 0,C 180,E1 13521.658,E2 13521.658} C_VEL
LIN {X 0,Y 440.981,Z 992.213,A -85,B 0,C 180,E1 13520.747,E2 13520.747} C_VEL
LIN {X 0,Y 447.197,Z 971.069,A -85,B 0,C 180,E1 13520.035,E2 13520.035} C_VEL
LIN {X 0,Y 452.549,Z 949.872,A -85,B 0,C 180,E1 13519.445,E2 13519.445} C_VEL
LIN {X 0,Y 457.381,Z 926.954,A -85,B 0,C 180,E1 13518.935,E2 13518.935} C_VEL
LIN {X 0,Y 462.07,Z 896.324,A -85,B 0,C 180,E1 13518.377,E2 13518.377} C_VEL
LIN {X 0,Y 467.968,Z 833.407,A -85,B 0,C 180,E1 13517.409,E2 13517.409} C_VEL
LIN {X 0,Y 484.673,Z 650.387,A -85,B 0,C 180,E1 13514.645,E2 13514.645} C_VEL
LIN {X 0,Y 480.935,Z 642.75,A -85,B 0,C 180,E1 13512.365,E2 13512.365} C_VEL
LIN {X 0,Y 477.867,Z 637.527,A -85,B 0,C 180,E1 13510.184,E2 13510.184} C_VEL
LIN {X 0,Y 476.124,Z 634.537,A -85,B 0,C 180,E1 13508.697,E2 13508.697} C_VEL
LIN {X 0,Y 473.72,Z 630.285,A -85,B 0,C 180,E1 13506.058,E2 13506.058} C_VEL
LIN {X 0,Y 471.734,Z 626.562,A -85,B 0,C 180,E1 13502.187,E2 13502.187} C_VEL
LIN {X 0,Y 471.574,Z 625.441,A -85,B 0,C 180,E1 13501.093,E2 13501.093} C_VEL
LIN {X 0,Y 471.625,Z 625.636,A -85,B 0,C 180,E1 13498.056,E2 13498.056} C_VEL
LIN {X 0,Y 473.243,Z 629.774,A -85,B 0,C 180,E1 13494.057,E2 13494.057} C_VEL
LIN {X 0,Y 474.085,Z 630.881,A -85,B 0,C 180,E1 13492.973,E2 13492.973} C_VEL
LIN {X 0,Y 476.913,Z 635.816,A -85,B 0,C 180,E1 13490.1,E2 13490.1} C_VEL
LIN {X 0,Y 479.763,Z 640.777,A -85,B 0,C 180,E1 13487.909,E2 13487.909} C_VEL
LIN {X 0,Y 483.303,Z 646.779,A -85,B 0,C 180,E1 13485.686,E2 13485.686} C_VEL
LIN {X 0,Y 484.579,Z 649.336,A -85,B 0,C 180,E1 13484.95,E2 13484.95} C_VEL
LIN {X 0,Y 464.31,Z 871.287,A -85,B 0,C 180,E1 13481.616,E2 13481.616} C_VEL
LIN {X 0,Y 460.923,Z 899.318,A -85,B 0,C 180,E1 13481.152,E2 13481.152} C_VEL
LIN {X 0,Y 457.162,Z 921.384,A -85,B 0,C 180,E1 13480.709,E2 13480.709} C_VEL
LIN {X 0,Y 452.603,Z 942.873,A -85,B 0,C 180,E1 13480.167,E2 13480.167} C_VEL
LIN {X 0,Y 446.585,Z 966.452,A -85,B 0,C 180,E1 13479.438,E2 13479.438} C_VEL
LIN {X 0,Y 438.593,Z 992.442,A -85,B 0,C 180,E1 13478.433,E2 13478.433} C_VEL
LIN {X 0,Y 430.902,Z 1013.954,A -85,B 0,C 180,E1 13477.425,E2 13477.425} C_VEL
LIN {X 0,Y 423.354,Z 1032.893,A -85,B 0,C 180,E1 13476.381,E2 13476.381} C_VEL
LIN {X 0,Y 414.832,Z 1052.261,A -85,B 0,C 180,E1 13475.139,E2 13475.139} C_VEL
LIN {X 0,Y 404.022,Z 1074.697,A -85,B 0,C 180,E1 13473.443,E2 13473.443} C_VEL
LIN {X 0,Y 392.151,Z 1096.653,A -85,B 0,C 180,E1 13471.429,E2 13471.429} C_VEL
LIN {X 0,Y 382.423,Z 1113.416,A -85,B 0,C 180,E1 13469.616,E2 13469.616} C_VEL
LIN {X 0,Y 372.741,Z 1129.1,A -85,B 0,C 180,E1 13467.653,E2 13467.653} C_VEL
LIN {X 0,Y 362.291,Z 1145.154,A -85,B 0,C 180,E1 13465.313,E2 13465.313} C_VEL
LIN {X 0,Y 349.114,Z 1164.33,A -85,B 0,C 180,E1 13461.947,E2 13461.947} C_VEL
LIN {X 0,Y 339.09,Z 1178.251,A -85,B 0,C 180,E1 13458.999,E2 13458.999} C_VEL
LIN {X 0,Y 330.393,Z 1190.09,A -85,B 0,C 180,E1 13456.062,E2 13456.062} C_VEL
LIN {X 0,Y 322.069,Z 1201.285,A -85,B 0,C 180,E1 13452.822,E2 13452.822} C_VEL
LIN {X 0,Y 313.226,Z 1213.267,A -85,B 0,C 180,E1 13448.718,E2 13448.718} C_VEL
LIN {X 0,Y 304.953,Z 1224.698,A -85,B 0,C 180,E1 13443.864,E2 13443.864} C_VEL
LIN {X 0,Y 299.591,Z 1232.569,A -85,B 0,C 180,E1 13439.801,E2 13439.801} C_VEL
LIN {X 0,Y 295.402,Z 1239.255,A -85,B 0,C 180,E1 13435.663,E2 13435.663} C_VEL
LIN {X 0,Y 292.147,Z 1245.094,A -85,B 0,C 180,E1 13431.261,E2 13431.261} C_VEL
LIN {X 0,Y 289.701,Z 1250.57,A -85,B 0,C 180,E1 13426.018,E2 13426.018} C_VEL
LIN {X 0,Y 288.505,Z 1254.192,A -85,B 0,C 180,E1 13420.979,E2 13420.979} C_VEL
LIN {X 0,Y 288.118,Z 1256.277,A -85,B 0,C 180,E1 13416.567,E2 13416.567} C_VEL
LIN {X 0,Y 288.003,Z 1257.277,A -85,B 0,C 180,E1 13412.578,E2 13412.578} C_VEL
LIN {X 0,Y 287.98,Z 1257.417,A -85,B 0,C 180,E1 13408.598,E2 13408.598} C_VEL
LIN {X 0,Y 288.056,Z 1256.696,A -85,B 0,C 180,E1 13404.613,E2 13404.613} C_VEL
LIN {X 0,Y 288.306,Z 1255.109,A -85,B 0,C 180,E1 13400.61,E2 13400.61} C_VEL
LIN {X 0,Y 289.003,Z 1252.486,A -85,B 0,C 180,E1 13396.384,E2 13396.384} C_VEL
LIN {X 0,Y 290.385,Z 1248.866,A -85,B 0,C 180,E1 13392.146,E2 13392.146} C_VEL
LIN {X 0,Y 292.62,Z 1244.216,A -85,B 0,C 180,E1 13387.913,E2 13387.913} C_VEL
LIN {X 0,Y 296.068,Z 1238.19,A -85,B 0,C 180,E1 13383.505,E2 13383.505} C_VEL
LIN {X 0,Y 301.944,Z 1229.198,A -85,B 0,C 180,E1 13378.221,E2 13378.221} C_VEL
LIN {X 0,Y 308.777,Z 1219.369,A -85,B 0,C 180,E1 13373.651,E2 13373.651} C_VEL
LIN {X 0,Y 315.68,Z 1209.941,A -85,B 0,C 180,E1 13369.977,E2 13369.977} C_VEL
LIN {X 0,Y 323.626,Z 1199.257,A -85,B 0,C 180,E1 13366.442,E2 13366.442} C_VEL
LIN {X 0,Y 334.064,Z 1185.329,A -85,B 0,C 180,E1 13362.567,E2 13362.567} C_VEL
LIN {X 0,Y 345.194,Z 1169.922,A -85,B 0,C 180,E1 13359.07,E2 13359.07} C_VEL
LIN {X 0,Y 355.136,Z 1155.767,A -85,B 0,C 180,E1 13356.359,E2 13356.359} C_VEL
LIN {X 0,Y 365.168,Z 1140.927,A -85,B 0,C 180,E1 13353.928,E2 13353.928} C_VEL
LIN {X 0,Y 376.436,Z 1123.46,A -85,B 0,C 180,E1 13351.492,E2 13351.492} C_VEL
LIN {X 0,Y 388.963,Z 1102.498,A -85,B 0,C 180,E1 13349.063,E2 13349.063} C_VEL
LIN {X 0,Y 399.02,Z 1084.32,A -85,B 0,C 180,E1 13347.295,E2 13347.295} C_VEL
LIN {X 0,Y 406.768,Z 1069.37,A -85,B 0,C 180,E1 13346.033,E2 13346.033} C_VEL
LIN {X 0,Y 409.324,Z 1063.395,A -85,B 0,C 180,E1 13345.442,E2 13345.442} C_VEL
LIN {X 0,Y 414.138,Z 1047.948,A -85,B 0,C 180,E1 13343.526,E2 13343.526} C_VEL
LIN {X 0,Y 416.305,Z 1042.588,A -85,B 0,C 180,E1 13343.075,E2 13343.075} C_VEL
LIN {X 0,Y 426.215,Z 1018.864,A -85,B 0,C 180,E1 13341.711,E2 13341.711} C_VEL
LIN {X 0,Y 433.624,Z 999.053,A -85,B 0,C 180,E1 13340.758,E2 13340.758} C_VEL
LIN {X 0,Y 440.528,Z 978.202,A -85,B 0,C 180,E1 13339.905,E2 13339.905} C_VEL
LIN {X 0,Y 446.534,Z 957.355,A -85,B 0,C 180,E1 13339.189,E2 13339.189} C_VEL
LIN {X 0,Y 452.974,Z 930.82,A -85,B 0,C 180,E1 13338.45,E2 13338.45} C_VEL
LIN {X 0,Y 457.773,Z 904.679,A -85,B 0,C 180,E1 13337.895,E2 13337.895} C_VEL
LIN {X 0,Y 460.835,Z 882.322,A -85,B 0,C 180,E1 13337.515,E2 13337.515} C_VEL
LIN {X 0,Y 480.818,Z 669.854,A -85,B 0,C 180,E1 13334.334,E2 13334.334} C_VEL
LIN {X 0,Y 482.217,Z 654.942,A -85,B 0,C 180,E1 13334.102,E2 13334.102} C_VEL
LIN {X 0,Y 478.833,Z 648.949,A -85,B 0,C 180,E1 13331.931,E2 13331.931} C_VEL
LIN {X 0,Y 476.72,Z 645.255,A -85,B 0,C 180,E1 13330.331,E2 13330.331} C_VEL
LIN {X 0,Y 475.046,Z 642.254,A -85,B 0,C 180,E1 13328.839,E2 13328.839} C_VEL
LIN {X 0,Y 472.751,Z 638.117,A -85,B 0,C 180,E1 13326.192,E2 13326.192} C_VEL
LIN {X 0,Y 470.886,Z 634.092,A -85,B 0,C 180,E1 13321.947,E2 13321.947} C_VEL
LIN {X 0,Y 470.81,Z 633.408,A -85,B 0,C 180,E1 13321.095,E2 13321.095} C_VEL
LIN {X 0,Y 470.864,Z 633.694,A -85,B 0,C 180,E1 13318.783,E2 13318.783} C_VEL
LIN {X 0,Y 472.346,Z 637.711,A -85,B 0,C 180,E1 13314.777,E2 13314.777} C_VEL
LIN {X 0,Y 473.196,Z 638.882,A -85,B 0,C 180,E1 13313.631,E2 13313.631} C_VEL
LIN {X 0,Y 475.946,Z 643.803,A -85,B 0,C 180,E1 13310.752,E2 13310.752} C_VEL
LIN {X 0,Y 478.566,Z 648.508,A -85,B 0,C 180,E1 13308.674,E2 13308.674} C_VEL
LIN {X 0,Y 480.56,Z 652.157,A -85,B 0,C 180,E1 13307.32,E2 13307.32} C_VEL
LIN {X 0,Y 482.327,Z 656.224,A -85,B 0,C 180,E1 13306.185,E2 13306.185} C_VEL
LIN {X 0,Y 462.076,Z 873.915,A -85,B 0,C 180,E1 13302.93,E2 13302.93} C_VEL
LIN {X 0,Y 458.257,Z 907.272,A -85,B 0,C 180,E1 13302.391,E2 13302.391} C_VEL
LIN {X 0,Y 454.264,Z 930.354,A -85,B 0,C 180,E1 13301.958,E2 13301.958} C_VEL
LIN {X 0,Y 449.507,Z 952.047,A -85,B 0,C 180,E1 13301.471,E2 13301.471} C_VEL
LIN {X 0,Y 443.561,Z 974.752,A -85,B 0,C 180,E1 13300.834,E2 13300.834} C_VEL
LIN {X 0,Y 434.958,Z 1002.19,A -85,B 0,C 180,E1 13299.865,E2 13299.865} C_VEL
LIN {X 0,Y 426.937,Z 1024.131,A -85,B 0,C 180,E1 13298.903,E2 13298.903} C_VEL
LIN {X 0,Y 418.83,Z 1043.994,A -85,B 0,C 180,E1 13297.872,E2 13297.872} C_VEL
LIN {X 0,Y 410.014,Z 1063.645,A -85,B 0,C 180,E1 13296.667,E2 13296.667} C_VEL
LIN {X 0,Y 398.432,Z 1087.142,A -85,B 0,C 180,E1 13294.96,E2 13294.96} C_VEL
LIN {X 0,Y 386.506,Z 1108.807,A -85,B 0,C 180,E1 13293.035,E2 13293.035} C_VEL
LIN {X 0,Y 376.421,Z 1125.929,A -85,B 0,C 180,E1 13291.241,E2 13291.241} C_VEL
LIN {X 0,Y 366.083,Z 1142.501,A -85,B 0,C 180,E1 13289.213,E2 13289.213} C_VEL
LIN {X 0,Y 353.75,Z 1161.288,A -85,B 0,C 180,E1 13286.502,E2 13286.502} C_VEL
LIN {X 0,Y 341.356,Z 1178.998,A -85,B 0,C 180,E1 13283.387,E2 13283.387} C_VEL
LIN {X 0,Y 331.19,Z 1193.11,A -85,B 0,C 180,E1 13280.429,E2 13280.429} C_VEL
LIN {X 0,Y 321.615,Z 1206.177,A -85,B 0,C 180,E1 13277.207,E2 13277.207} C_VEL
LIN {X 0,Y 311.08,Z 1220.618,A -85,B 0,C 180,E1 13272.963,E2 13272.963} C_VEL
LIN {X 0,Y 302.078,Z 1232.913,A -85,B 0,C 180,E1 13268.492,E2 13268.492} C_VEL
LIN {X 0,Y 295.584,Z 1242.309,A -85,B 0,C 180,E1 13264.405,E2 13264.405} C_VEL
LIN {X 0,Y 290.286,Z 1250.512,A -85,B 0,C 180,E1 13260.166,E2 13260.166} C_VEL
LIN {X 0,Y 285.641,Z 1258.669,A -85,B 0,C 180,E1 13255.068,E2 13255.068} C_VEL
LIN {X 0,Y 282.341,Z 1265.6,A -85,B 0,C 180,E1 13249.453,E2 13249.453} C_VEL
LIN {X 0,Y 280.836,Z 1269.942,A -85,B 0,C 180,E1 13244.862,E2 13244.862} C_VEL
LIN {X 0,Y 280.181,Z 1272.889,A -85,B 0,C 180,E1 13240.703,E2 13240.703} C_VEL
LIN {X 0,Y 280.004,Z 1274.884,A -85,B 0,C 180,E1 13236.571,E2 13236.571} C_VEL
LIN {X 0,Y 279.99,Z 1275.905,A -85,B 0,C 180,E1 13232.67,E2 13232.67} C_VEL
LIN {X 0,Y 279.975,Z 1276.071,A -85,B 0,C 180,E1 13228.782,E2 13228.782} C_VEL
LIN {X 0,Y 279.986,Z 1275.313,A -85,B 0,C 180,E1 13224.682,E2 13224.682} C_VEL
LIN {X 0,Y 280.073,Z 1273.603,A -85,B 0,C 180,E1 13220.558,E2 13220.558} C_VEL
LIN {X 0,Y 280.618,Z 1270.777,A -85,B 0,C 180,E1 13216.199,E2 13216.199} C_VEL
LIN {X 0,Y 281.828,Z 1266.892,A -85,B 0,C 180,E1 13211.818,E2 13211.818} C_VEL
LIN {X 0,Y 283.917,Z 1261.926,A -85,B 0,C 180,E1 13207.438,E2 13207.438} C_VEL
LIN {X 0,Y 286.921,Z 1256.166,A -85,B 0,C 180,E1 13203.297,E2 13203.297} C_VEL
LIN {X 0,Y 291.436,Z 1248.636,A -85,B 0,C 180,E1 13198.81,E2 13198.81} C_VEL
LIN {X 0,Y 298.505,Z 1238.088,A -85,B 0,C 180,E1 13193.651,E2 13193.651} C_VEL
LIN {X 0,Y 306.71,Z 1226.417,A -85,B 0,C 180,E1 13189.074,E2 13189.074} C_VEL
LIN {X 0,Y 314.786,Z 1215.355,A -85,B 0,C 180,E1 13185.428,E2 13185.428} C_VEL
LIN {X 0,Y 323.476,Z 1203.576,A -85,B 0,C 180,E1 13182.126,E2 13182.126} C_VEL
LIN {X 0,Y 335.299,Z 1187.514,A -85,B 0,C 180,E1 13178.336,E2 13178.336} C_VEL
LIN {X 0,Y 347.076,Z 1170.754,A -85,B 0,C 180,E1 13175.115,E2 13175.115} C_VEL
LIN {X 0,Y 357.392,Z 1155.617,A -85,B 0,C 180,E1 13172.654,E2 13172.654} C_VEL
LIN {X 0,Y 367.465,Z 1140.179,A -85,B 0,C 180,E1 13170.501,E2 13170.501} C_VEL
LIN {X 0,Y 377.718,Z 1123.624,A -85,B 0,C 180,E1 13168.515,E2 13168.515} C_VEL
LIN {X 0,Y 390.513,Z 1101.594,A -85,B 0,C 180,E1 13166.293,E2 13166.293} C_VEL
LIN {X 0,Y 401.655,Z 1080.422,A -85,B 0,C 180,E1 13164.534,E2 13164.534} C_VEL
LIN {X 0,Y 411.061,Z 1061.074,A -85,B 0,C 180,E1 13163.175,E2 13163.175} C_VEL
LIN {X 0,Y 419.518,Z 1042.054,A -85,B 0,C 180,E1 13162.03,E2 13162.03} C_VEL
LIN {X 0,Y 428.521,Z 1019.726,A -85,B 0,C 180,E1 13160.896,E2 13160.896} C_VEL
LIN {X 0,Y 437.768,Z 993.23,A -85,B 0,C 180,E1 13159.801,E2 13159.801} C_VEL
LIN {X 0,Y 444.284,Z 971.538,A -85,B 0,C 180,E1 13159.077,E2 13159.077} C_VEL
LIN {X 0,Y 449.772,Z 950.246,A -85,B 0,C 180,E1 13158.492,E2 13158.492} C_VEL
LIN {X 0,Y 454.571,Z 927.984,A -85,B 0,C 180,E1 13158.002,E2 13158.002} C_VEL
LIN {X 0,Y 459.165,Z 899.873,A -85,B 0,C 180,E1 13157.486,E2 13157.486} C_VEL
LIN {X 0,Y 463.759,Z 853.517,A -85,B 0,C 180,E1 13156.77,E2 13156.77} C_VEL
LIN {X 0,Y 482.167,Z 655.869,A -85,B 0,C 180,E1 13153.814,E2 13153.814} C_VEL
LIN {X 0,Y 479.399,Z 650.159,A -85,B 0,C 180,E1 13152.039,E2 13152.039} C_VEL
LIN {X 0,Y 476.433,Z 644.963,A -85,B 0,C 180,E1 13149.849,E2 13149.849} C_VEL
LIN {X 0,Y 474.88,Z 642.25,A -85,B 0,C 180,E1 13148.476,E2 13148.476} C_VEL
LIN {X 0,Y 472.649,Z 638.167,A -85,B 0,C 180,E1 13145.95,E2 13145.95} C_VEL
LIN {X 0,Y 470.726,Z 634.442,A -85,B 0,C 180,E1 13142.069,E2 13142.069} C_VEL
LIN {X 0,Y 470.577,Z 633.385,A -85,B 0,C 180,E1 13140.974,E2 13140.974} C_VEL
LIN {X 0,Y 470.629,Z 633.52,A -85,B 0,C 180,E1 13138.174,E2 13138.174} C_VEL
LIN {X 0,Y 472.182,Z 637.654,A -85,B 0,C 180,E1 13134.166,E2 13134.166} C_VEL
LIN {X 0,Y 473.047,Z 638.916,A -85,B 0,C 180,E1 13133.019,E2 13133.019} C_VEL
LIN {X 0,Y 475.716,Z 643.644,A -85,B 0,C 180,E1 13130.259,E2 13130.259} C_VEL
LIN {X 0,Y 478.515,Z 648.624,A -85,B 0,C 180,E1 13128.061,E2 13128.061} C_VEL
LIN {X 0,Y 481.898,Z 654.534,A -85,B 0,C 180,E1 13125.889,E2 13125.889} C_VEL
LIN {X 0,Y 482.037,Z 655.099,A -85,B 0,C 180,E1 13125.788,E2 13125.788} C_VEL
LIN {X 0,Y 461.335,Z 876.37,A -85,B 0,C 180,E1 13122.483,E2 13122.483} C_VEL
